LIN {X 0.035,Y -406.646,Z 971.492,A 0.000,B 0.000,C 90.000,E1 268.568} C_DIS
LIN {X -0.087,Y -402.210,Z 971.492,A 0.000,B 0.000,C 90.000,E1 268.568} C_DIS
LIN {X -0.066,Y -181.223,Z 971.492,A 0.000,B 0.000,C 90.000,E1 268.568} C_DIS
LIN {X 0.036,Y -180.887,Z 971.473,A 0.000,B 0.000,C 90.000,E1 265.122} C_DIS
LIN {X -0.082,Y -179.009,Z 971.445,A 0.000,B 0.000,C 90.000,E1 260.095} C_DIS
LIN {X 0.013,Y -178.623,Z 971.440,A 0.000,B 0.000,C 90.000,E1 259.218} C_DIS
LIN {X -0.088,Y -175.674,Z 971.412,A 0.000,B 0.000,C 90.000,E1 254.157} C_DIS
LIN {X -0.076,Y -172.391,Z 971.388,A 0.000,B 0.000,C 90.000,E1 249.880} C_DIS
LIN {X -0.060,Y -171.196,Z 971.379,A 0.000,B 0.000,C 90.000,E1 248.156} C_DIS
LIN {X -0.008,Y -167.485,Z 971.355,A 0.000,B 0.000,C 90.000,E1 243.819} C_DIS
LIN {X 0.000,Y -166.882,Z 971.350,A 0.000,B 0.000,C 90.000,E1 242.948} C_DIS
LIN {X -0.009,Y -162.187,Z 971.321,A 0.000,B 0.000,C 90.000,E1 237.709} C_DIS
LIN {X -0.042,Y -160.756,Z 971.311,A 0.000,B 0.000,C 90.000,E1 235.960} C_DIS
LIN {X 0.027,Y -157.553,Z 971.291,A 0.000,B 0.000,C 90.000,E1 232.396} C_DIS
LIN {X -0.035,Y -155.582,Z 971.276,A 0.000,B 0.000,C 90.000,E1 229.747} C_DIS
LIN {X 0.017,Y -151.866,Z 971.251,A 0.000,B 0.000,C 90.000,E1 225.243} C_DIS
LIN {X 0.030,Y -150.090,Z 971.236,A 0.000,B 0.000,C 90.000,E1 222.528} C_DIS
LIN {X -0.052,Y -146.891,Z 971.211,A 0.000,B 0.000,C 90.000,E1 218.016} C_DIS
LIN {X 0.053,Y -145.478,Z 971.196,A 0.000,B 0.000,C 90.000,E1 215.231} C_DIS
LIN {X -0.031,Y -142.888,Z 971.170,A 0.000,B 0.000,C 90.000,E1 210.669} C_DIS
LIN {X 0.026,Y -141.507,Z 971.150,A 0.000,B 0.000,C 90.000,E1 206.950} C_DIS
LIN {X -0.056,Y -139.391,Z 971.114,A 0.000,B 0.000,C 90.000,E1 200.482} C_DIS
LIN {X -0.005,Y -139.098,Z 971.103,A 0.000,B 0.000,C 90.000,E1 198.598} C_DIS
LIN {X -0.014,Y -138.353,Z 971.057,A 0.000,B 0.000,C 90.000,E1 190.197} C_DIS
LIN {X -0.020,Y -139.515,Z 971.005,A 0.000,B 0.000,C 90.000,E1 180.859} C_DIS
LIN {X 0.060,Y -141.167,Z 970.974,A 0.000,B 0.000,C 90.000,E1 175.241} C_DIS
LIN {X 0.032,Y -142.546,Z 970.958,A 0.000,B 0.000,C 90.000,E1 172.470} C_DIS
LIN {X -0.042,Y -144.821,Z 970.933,A 0.000,B 0.000,C 90.000,E1 167.881} C_DIS
LIN {X -0.056,Y -147.443,Z 970.912,A 0.000,B 0.000,C 90.000,E1 164.212} C_DIS
LIN {X -0.027,Y -150.023,Z 970.892,A 0.000,B 0.000,C 90.000,E1 160.550} C_DIS
LIN {X -0.021,Y -153.358,Z 970.872,A 0.000,B 0.000,C 90.000,E1 156.922} C_DIS
LIN {X 0.027,Y -155.892,Z 970.857,A 0.000,B 0.000,C 90.000,E1 154.204} C_DIS
LIN {X -0.075,Y -159.750,Z 970.837,A 0.000,B 0.000,C 90.000,E1 150.667} C_DIS
LIN {X -0.009,Y -161.990,Z 970.827,A 0.000,B 0.000,C 90.000,E1 148.869} C_DIS
LIN {X 0.011,Y -166.182,Z 970.807,A 0.000,B 0.000,C 90.000,E1 145.341} C_DIS
LIN {X 0.003,Y -171.197,Z 970.788,A 0.000,B 0.000,C 90.000,E1 141.859} C_DIS
LIN {X 0.033,Y -176.080,Z 970.769,A 0.000,B 0.000,C 90.000,E1 138.405} C_DIS
LIN {X -0.104,Y -180.340,Z 970.755,A 0.000,B 0.000,C 90.000,E1 135.891} C_DIS
LIN {X 0.004,Y -185.750,Z 970.736,A 0.000,B 0.000,C 90.000,E1 132.486} C_DIS
LIN {X -0.082,Y -190.362,Z 970.722,A 0.000,B 0.000,C 90.000,E1 130.011} C_DIS
LIN {X -0.069,Y -195.145,Z 970.707,A 0.000,B 0.000,C 90.000,E1 127.237} C_DIS
LIN {X -0.152,Y -298.444,Z 970.707,A 0.000,B 0.000,C 90.000,E1 127.237} C_DIS
LIN {X 0.125,Y -300.189,Z 970.707,A 0.000,B 0.000,C 90.000,E1 127.156} C_DIS
LIN {X -0.078,Y -305.216,Z 970.705,A 0.000,B 0.000,C 90.000,E1 126.950} C_DIS
LIN {X 0.147,Y -307.899,Z 970.704,A 0.000,B 0.000,C 90.000,E1 126.664} C_DIS
LIN {X -0.023,Y -311.652,Z 970.701,A 0.000,B 0.000,C 90.000,E1 126.171} C_DIS
LIN {X -0.057,Y -313.281,Z 970.699,A 0.000,B 0.000,C 90.000,E1 125.851} C_DIS
LIN {X -0.020,Y -314.559,Z 970.697,A 0.000,B 0.000,C 90.000,E1 125.518} C_DIS
LIN {X -0.088,Y -326.270,Z 970.678,A 0.000,B 0.000,C 90.000,E1 122.005} C_DIS
LIN {X 0.038,Y -337.255,Z 970.662,A 0.000,B 0.000,C 90.000,E1 119.155} C_DIS
LIN {X 0.165,Y -349.630,Z 970.647,A 0.000,B 0.000,C 90.000,E1 116.360} C_DIS
LIN {X 0.178,Y -363.508,Z 970.632,A 0.000,B 0.000,C 90.000,E1 113.643} C_DIS
LIN {X 0.187,Y -377.204,Z 970.618,A 0.000,B 0.000,C 90.000,E1 111.280} C_DIS
LIN {X -0.107,Y -392.279,Z 970.606,A 0.000,B 0.000,C 90.000,E1 109.014} C_DIS
LIN {X 0.084,Y -408.843,Z 970.593,A 0.000,B 0.000,C 90.000,E1 106.732} C_DIS
LIN {X 0.073,Y -427.015,Z 970.581,A 0.000,B 0.000,C 90.000,E1 104.537} C_DIS
LIN {X 0.151,Y -446.708,Z 970.569,A 0.000,B 0.000,C 90.000,E1 102.411} C_DIS
LIN {X -0.068,Y -467.052,Z 970.558,A 0.000,B 0.000,C 90.000,E1 100.489} C_DIS
LIN {X -0.062,Y -469.165,Z 970.557,A 0.000,B 0.000,C 90.000,E1 100.254} C_DIS
LIN {X -0.057,Y -470.766,Z 970.556,A 0.000,B 0.000,C 90.000,E1 100.018} C_DIS
LIN {X 0.261,Y -472.078,Z 970.554,A 0.000,B 0.000,C 90.000,E1 99.726} C_DIS
LIN {X 0.034,Y -473.047,Z 970.553,A 0.000,B 0.000,C 90.000,E1 99.500} C_DIS
LIN {X 0.219,Y -474.135,Z 970.550,A 0.000,B 0.000,C 90.000,E1 98.973} C_DIS
LIN {X -0.132,Y -474.233,Z 970.547,A 0.000,B 0.000,C 90.000,E1 98.511} C_DIS
LIN {X -0.007,Y -473.359,Z 970.544,A 0.000,B 0.000,C 90.000,E1 97.992} C_DIS
LIN {X 0.121,Y -471.370,Z 970.542,A 0.000,B 0.000,C 90.000,E1 97.473} C_DIS
LIN {X -0.164,Y -468.113,Z 970.539,A 0.000,B 0.000,C 90.000,E1 97.004} C_DIS
LIN {X 0.071,Y -454.642,Z 970.527,A 0.000,B 0.000,C 90.000,E1 94.935} C_DIS
LIN {X -0.006,Y -441.028,Z 970.516,A 0.000,B 0.000,C 90.000,E1 92.865} C_DIS
LIN {X 0.133,Y -426.286,Z 970.503,A 0.000,B 0.000,C 90.000,E1 90.458} C_DIS
LIN {X -0.094,Y -412.655,Z 970.489,A 0.000,B 0.000,C 90.000,E1 88.051} C_DIS
LIN {X -0.026,Y -403.632,Z 970.480,A 0.000,B 0.000,C 90.000,E1 86.388} C_DIS
LIN {X -0.040,Y -392.927,Z 970.469,A 0.000,B 0.000,C 90.000,E1 84.432} C_DIS
LIN {X 0.117,Y -383.619,Z 970.460,A 0.000,B 0.000,C 90.000,E1 82.704} C_DIS
LIN {X 0.192,Y -375.672,Z 970.452,A 0.000,B 0.000,C 90.000,E1 81.254} C_DIS
LIN {X 0.119,Y -364.228,Z 970.440,A 0.000,B 0.000,C 90.000,E1 79.218} C_DIS
LIN {X -0.119,Y -352.438,Z 970.429,A 0.000,B 0.000,C 90.000,E1 77.173} C_DIS
LIN {X 0.005,Y -334.406,Z 970.410,A 0.000,B 0.000,C 90.000,E1 73.795} C_DIS
LIN {X 0.084,Y -322.122,Z 970.396,A 0.000,B 0.000,C 90.000,E1 71.275} C_DIS
LIN {X -0.148,Y -311.513,Z 970.384,A 0.000,B 0.000,C 90.000,E1 69.082} C_DIS
LIN {X 0.077,Y -299.564,Z 970.369,A 0.000,B 0.000,C 90.000,E1 66.433} C_DIS
LIN {X 0.082,Y -287.783,Z 970.354,A 0.000,B 0.000,C 90.000,E1 63.768} C_DIS
LIN {X 0.102,Y -277.508,Z 970.341,A 0.000,B 0.000,C 90.000,E1 61.385} C_DIS
LIN {X 0.083,Y -266.012,Z 970.326,A 0.000,B 0.000,C 90.000,E1 58.614} C_DIS
LIN {X -0.021,Y -254.922,Z 970.310,A 0.000,B 0.000,C 90.000,E1 55.801} C_DIS
LIN {X -0.099,Y -243.035,Z 970.292,A 0.000,B 0.000,C 90.000,E1 52.557} C_DIS
LIN {X 0.074,Y -232.031,Z 970.273,A 0.000,B 0.000,C 90.000,E1 49.175} C_DIS
LIN {X -0.120,Y -221.821,Z 970.254,A 0.000,B 0.000,C 90.000,E1 45.810} C_DIS
LIN {X -0.005,Y -213.311,Z 970.237,A 0.000,B 0.000,C 90.000,E1 42.690} C_DIS
LIN {X -0.070,Y -205.336,Z 970.220,A 0.000,B 0.000,C 90.000,E1 39.564} C_DIS
LIN {X -0.111,Y -197.993,Z 970.202,A 0.000,B 0.000,C 90.000,E1 36.377} C_DIS
LIN {X 0.027,Y -191.300,Z 970.184,A 0.000,B 0.000,C 90.000,E1 33.086} C_DIS
LIN {X 0.004,Y -185.309,Z 970.166,A 0.000,B 0.000,C 90.000,E1 29.795} C_DIS
LIN {X 0.049,Y -180.063,Z 970.147,A 0.000,B 0.000,C 90.000,E1 26.437} C_DIS
LIN {X -0.026,Y -175.534,Z 970.128,A 0.000,B 0.000,C 90.000,E1 23.078} C_DIS
LIN {X 0.064,Y -171.707,Z 970.109,A 0.000,B 0.000,C 90.000,E1 19.631} C_DIS
LIN {X -0.096,Y -167.927,Z 970.085,A 0.000,B 0.000,C 90.000,E1 15.371} C_DIS
LIN {X -0.056,Y -165.174,Z 970.061,A 0.000,B 0.000,C 90.000,E1 11.007} C_DIS
LIN {X -0.067,Y -163.070,Z 970.027,A 0.000,B 0.000,C 90.000,E1 4.878} C_DIS
LIN {X -0.042,Y -164.371,Z 969.963,A 0.000,B 0.000,C 90.000,E1 353.394} C_DIS
LIN {X 0.037,Y -167.337,Z 969.934,A 0.000,B 0.000,C 90.000,E1 348.117} C_DIS
LIN {X 0.069,Y -170.198,Z 969.915,A 0.000,B 0.000,C 90.000,E1 344.629} C_DIS
LIN {X -0.066,Y -173.819,Z 969.896,A 0.000,B 0.000,C 90.000,E1 341.221} C_DIS
LIN {X -0.058,Y -178.179,Z 969.877,A 0.000,B 0.000,C 90.000,E1 337.794} C_DIS
LIN {X -0.067,Y -183.323,Z 969.858,A 0.000,B 0.000,C 90.000,E1 334.409} C_DIS
LIN {X -0.037,Y -189.184,Z 969.839,A 0.000,B 0.000,C 90.000,E1 331.051} C_DIS
LIN {X -0.009,Y -195.645,Z 969.821,A 0.000,B 0.000,C 90.000,E1 327.740} C_DIS
LIN {X -0.001,Y -202.711,Z 969.803,A 0.000,B 0.000,C 90.000,E1 324.482} C_DIS
LIN {X -0.010,Y -211.317,Z 969.783,A 0.000,B 0.000,C 90.000,E1 320.884} C_DIS
LIN {X -0.142,Y -220.576,Z 969.763,A 0.000,B 0.000,C 90.000,E1 317.391} C_DIS
LIN {X 0.031,Y -229.759,Z 969.746,A 0.000,B 0.000,C 90.000,E1 314.271} C_DIS
LIN {X 0.045,Y -237.519,Z 969.733,A 0.000,B 0.000,C 90.000,E1 312.000} C_DIS
LIN {X 0.047,Y -246.307,Z 969.721,A 0.000,B 0.000,C 90.000,E1 309.769} C_DIS
LIN {X 0.072,Y -254.422,Z 969.711,A 0.000,B 0.000,C 90.000,E1 307.935} C_DIS
LIN {X -0.038,Y -265.321,Z 969.699,A 0.000,B 0.000,C 90.000,E1 305.804} C_DIS
LIN {X -0.069,Y -281.207,Z 969.683,A 0.000,B 0.000,C 90.000,E1 303.007} C_DIS
LIN {X 0.092,Y -300.564,Z 969.666,A 0.000,B 0.000,C 90.000,E1 299.922} C_DIS
LIN {X -0.055,Y -314.475,Z 969.655,A 0.000,B 0.000,C 90.000,E1 297.975} C_DIS
LIN {X -0.079,Y -329.831,Z 969.645,A 0.000,B 0.000,C 90.000,E1 296.052} C_DIS
LIN {X -0.113,Y -354.177,Z 969.630,A 0.000,B 0.000,C 90.000,E1 293.387} C_DIS
LIN {X 0.029,Y -370.447,Z 969.621,A 0.000,B 0.000,C 90.000,E1 291.716} C_DIS
LIN {X 0.138,Y -389.009,Z 969.611,A 0.000,B 0.000,C 90.000,E1 289.885} C_DIS
LIN {X -0.209,Y -399.660,Z 969.605,A 0.000,B 0.000,C 90.000,E1 288.906} C_DIS
LIN {X 0.200,Y -409.889,Z 969.599,A 0.000,B 0.000,C 90.000,E1 287.819} C_DIS
LIN {X -0.155,Y -420.017,Z 969.593,A 0.000,B 0.000,C 90.000,E1 286.804} C_DIS
LIN {X -0.147,Y -429.751,Z 969.587,A 0.000,B 0.000,C 90.000,E1 285.717} C_DIS
LIN {X 0.255,Y -438.913,Z 969.581,A 0.000,B 0.000,C 90.000,E1 284.592} C_DIS
LIN {X -0.190,Y -447.466,Z 969.575,A 0.000,B 0.000,C 90.000,E1 283.592} C_DIS
LIN {X 0.160,Y -457.530,Z 969.568,A 0.000,B 0.000,C 90.000,E1 282.243} C_DIS
LIN {X -0.083,Y -465.137,Z 969.562,A 0.000,B 0.000,C 90.000,E1 281.243} C_DIS
LIN {X 0.128,Y -472.224,Z 969.557,A 0.000,B 0.000,C 90.000,E1 280.197} C_DIS
LIN {X 0.091,Y -476.879,Z 969.553,A 0.000,B 0.000,C 90.000,E1 279.443} C_DIS
LIN {X 0.100,Y -480.839,Z 969.548,A 0.000,B 0.000,C 90.000,E1 278.690} C_DIS
LIN {X 0.141,Y -484.221,Z 969.544,A 0.000,B 0.000,C 90.000,E1 277.936} C_DIS
LIN {X -0.093,Y -486.124,Z 969.541,A 0.000,B 0.000,C 90.000,E1 277.466} C_DIS
LIN {X 0.093,Y -487.737,Z 969.539,A 0.000,B 0.000,C 90.000,E1 276.947} C_DIS
LIN {X -0.193,Y -489.000,Z 969.536,A 0.000,B 0.000,C 90.000,E1 276.486} C_DIS
LIN {X 0.015,Y -489.957,Z 969.533,A 0.000,B 0.000,C 90.000,E1 275.967} C_DIS
LIN {X 0.184,Y -490.489,Z 969.530,A 0.000,B 0.000,C 90.000,E1 275.454} C_DIS
LIN {X -0.081,Y -490.737,Z 969.528,A 0.000,B 0.000,C 90.000,E1 274.992} C_DIS
LIN {X 0.144,Y -490.592,Z 969.525,A 0.000,B 0.000,C 90.000,E1 274.473} C_DIS
LIN {X -0.122,Y -489.956,Z 969.522,A 0.000,B 0.000,C 90.000,E1 274.012} C_DIS
LIN {X 0.067,Y -488.830,Z 969.519,A 0.000,B 0.000,C 90.000,E1 273.498} C_DIS
LIN {X -0.204,Y -487.113,Z 969.517,A 0.000,B 0.000,C 90.000,E1 273.037} C_DIS
LIN {X -0.022,Y -484.823,Z 969.514,A 0.000,B 0.000,C 90.000,E1 272.522} C_DIS
LIN {X 0.146,Y -481.691,Z 969.511,A 0.000,B 0.000,C 90.000,E1 272.007} C_DIS
LIN {X -0.166,Y -477.763,Z 969.508,A 0.000,B 0.000,C 90.000,E1 271.547} C_DIS
LIN {X -0.033,Y -472.805,Z 969.506,A 0.000,B 0.000,C 90.000,E1 271.031} C_DIS
LIN {X -0.206,Y -466.997,Z 969.503,A 0.000,B 0.000,C 90.000,E1 270.573} C_DIS
LIN {X 0.051,Y -460.783,Z 969.501,A 0.000,B 0.000,C 90.000,E1 270.115} C_DIS
LIN {X -0.192,Y -454.151,Z 969.499,A 0.000,B 0.000,C 90.000,E1 269.771} C_DIS
LIN {X 0.015,Y -447.184,Z 969.497,A 0.000,B 0.000,C 90.000,E1 269.427} C_DIS
LIN {X 0.193,Y -440.049,Z 969.495,A 0.000,B 0.000,C 90.000,E1 269.141} C_DIS
LIN {X -0.170,Y -432.430,Z 969.494,A 0.000,B 0.000,C 90.000,E1 268.969} C_DIS
LIN {X -0.149,Y -424.534,Z 969.493,A 0.000,B 0.000,C 90.000,E1 268.797} C_DIS
LIN {X 0.166,Y -416.590,Z 969.492,A 0.000,B 0.000,C 90.000,E1 268.625} C_DIS
LIN {X 0.033,Y -409.424,Z 969.492,A 0.000,B 0.000,C 90.000,E1 268.568} C_DIS
LIN {X -0.198,Y -403.286,Z 969.492,A 0.000,B 0.000,C 90.000,E1 268.568} C_DIS
LIN {X 0.068,Y -181.220,Z 969.492,A 0.000,B 0.000,C 90.000,E1 268.511} C_DIS
LIN {X -0.021,Y -180.884,Z 969.473,A 0.000,B 0.000,C 90.000,E1 265.122} C_DIS
LIN {X 0.039,Y -179.005,Z 969.445,A 0.000,B 0.000,C 90.000,E1 260.038} C_DIS
LIN {X -0.043,Y -178.610,Z 969.440,A 0.000,B 0.000,C 90.000,E1 259.218} C_DIS
LIN {X 0.026,Y -175.662,Z 969.412,A 0.000,B 0.000,C 90.000,E1 254.102} C_DIS
LIN {X 0.030,Y -172.379,Z 969.388,A 0.000,B 0.000,C 90.000,E1 249.826} C_DIS
LIN {X 0.044,Y -171.177,Z 969.378,A 0.000,B 0.000,C 90.000,E1 248.103} C_DIS
LIN {X 0.088,Y -167.472,Z 969.354,A 0.000,B 0.000,C 90.000,E1 243.768} C_DIS
LIN {X 0.021,Y -166.868,Z 969.350,A 0.000,B 0.000,C 90.000,E1 242.922} C_DIS
LIN {X 0.075,Y -162.173,Z 969.320,A 0.000,B 0.000,C 90.000,E1 237.661} C_DIS
LIN {X -0.005,Y -160.736,Z 969.311,A 0.000,B 0.000,C 90.000,E1 235.928} C_DIS
LIN {X -0.026,Y -157.538,Z 969.291,A 0.000,B 0.000,C 90.000,E1 232.396} C_DIS
LIN {X 0.032,Y -155.564,Z 969.276,A 0.000,B 0.000,C 90.000,E1 229.703} C_DIS
LIN {X -0.034,Y -151.853,Z 969.251,A 0.000,B 0.000,C 90.000,E1 225.243} C_DIS
LIN {X -0.020,Y -150.074,Z 969.236,A 0.000,B 0.000,C 90.000,E1 222.528} C_DIS
LIN {X 0.014,Y -146.880,Z 969.211,A 0.000,B 0.000,C 90.000,E1 217.971} C_DIS
LIN {X 0.003,Y -145.466,Z 969.196,A 0.000,B 0.000,C 90.000,E1 215.231} C_DIS
LIN {X -0.079,Y -142.879,Z 969.170,A 0.000,B 0.000,C 90.000,E1 210.669} C_DIS
LIN {X -0.023,Y -141.497,Z 969.150,A 0.000,B 0.000,C 90.000,E1 206.950} C_DIS
LIN {X 0.026,Y -139.387,Z 969.114,A 0.000,B 0.000,C 90.000,E1 200.429} C_DIS
LIN {X 0.014,Y -138.844,Z 969.098,A 0.000,B 0.000,C 90.000,E1 197.638} C_DIS
LIN {X -0.062,Y -138.353,Z 969.057,A 0.000,B 0.000,C 90.000,E1 190.197} C_DIS
LIN {X -0.070,Y -139.518,Z 969.005,A 0.000,B 0.000,C 90.000,E1 180.859} C_DIS
LIN {X 0.011,Y -141.176,Z 968.974,A 0.000,B 0.000,C 90.000,E1 175.241} C_DIS
LIN {X -0.017,Y -142.555,Z 968.958,A 0.000,B 0.000,C 90.000,E1 172.470} C_DIS
LIN {X 0.050,Y -144.833,Z 968.932,A 0.000,B 0.000,C 90.000,E1 167.825} C_DIS
LIN {X 0.036,Y -147.455,Z 968.912,A 0.000,B 0.000,C 90.000,E1 164.157} C_DIS
LIN {X -0.078,Y -150.039,Z 968.892,A 0.000,B 0.000,C 90.000,E1 160.550} C_DIS
LIN {X -0.072,Y -153.378,Z 968.872,A 0.000,B 0.000,C 90.000,E1 156.922} C_DIS
LIN {X -0.024,Y -155.910,Z 968.857,A 0.000,B 0.000,C 90.000,E1 154.204} C_DIS
LIN {X 0.090,Y -159.773,Z 968.837,A 0.000,B 0.000,C 90.000,E1 150.589} C_DIS
LIN {X -0.062,Y -162.014,Z 968.827,A 0.000,B 0.000,C 90.000,E1 148.869} C_DIS
LIN {X 0.052,Y -166.208,Z 968.807,A 0.000,B 0.000,C 90.000,E1 145.308} C_DIS
LIN {X 0.054,Y -171.223,Z 968.788,A 0.000,B 0.000,C 90.000,E1 141.823} C_DIS
LIN {X -0.022,Y -176.108,Z 968.769,A 0.000,B 0.000,C 90.000,E1 138.405} C_DIS
LIN {X 0.094,Y -180.372,Z 968.755,A 0.000,B 0.000,C 90.000,E1 135.810} C_DIS
LIN {X 0.072,Y -185.780,Z 968.736,A 0.000,B 0.000,C 90.000,E1 132.447} C_DIS
LIN {X 0.005,Y -190.396,Z 968.722,A 0.000,B 0.000,C 90.000,E1 129.967} C_DIS
LIN {X 0.030,Y -195.092,Z 968.707,A 0.000,B 0.000,C 90.000,E1 127.237} C_DIS
LIN {X -0.004,Y -298.842,Z 968.707,A 0.000,B 0.000,C 90.000,E1 127.237} C_DIS
LIN {X 0.000,Y -305.337,Z 968.705,A 0.000,B 0.000,C 90.000,E1 126.950} C_DIS
LIN {X 0.053,Y -308.226,Z 968.704,A 0.000,B 0.000,C 90.000,E1 126.664} C_DIS
LIN {X -0.047,Y -311.919,Z 968.701,A 0.000,B 0.000,C 90.000,E1 126.137} C_DIS
LIN {X -0.010,Y -313.464,Z 968.699,A 0.000,B 0.000,C 90.000,E1 125.804} C_DIS
LIN {X 0.028,Y -314.678,Z 968.697,A 0.000,B 0.000,C 90.000,E1 125.471} C_DIS
LIN {X 0.048,Y -325.248,Z 968.679,A 0.000,B 0.000,C 90.000,E1 122.260} C_DIS
LIN {X 0.145,Y -336.099,Z 968.664,A 0.000,B 0.000,C 90.000,E1 119.411} C_DIS
LIN {X -0.075,Y -348.336,Z 968.648,A 0.000,B 0.000,C 90.000,E1 116.668} C_DIS
LIN {X -0.110,Y -362.059,Z 968.633,A 0.000,B 0.000,C 90.000,E1 113.951} C_DIS
LIN {X -0.150,Y -375.608,Z 968.620,A 0.000,B 0.000,C 90.000,E1 111.589} C_DIS
LIN {X -0.124,Y -390.526,Z 968.607,A 0.000,B 0.000,C 90.000,E1 109.268} C_DIS
LIN {X 0.030,Y -406.921,Z 968.594,A 0.000,B 0.000,C 90.000,E1 106.985} C_DIS
LIN {X 0.091,Y -424.908,Z 968.582,A 0.000,B 0.000,C 90.000,E1 104.773} C_DIS
LIN {X 0.067,Y -444.470,Z 968.570,A 0.000,B 0.000,C 90.000,E1 102.647} C_DIS
LIN {X 0.155,Y -467.321,Z 968.558,A 0.000,B 0.000,C 90.000,E1 100.433} C_DIS
LIN {X 0.154,Y -469.373,Z 968.557,A 0.000,B 0.000,C 90.000,E1 100.197} C_DIS
LIN {X 0.152,Y -470.931,Z 968.555,A 0.000,B 0.000,C 90.000,E1 99.962} C_DIS
LIN {X 0.005,Y -472.201,Z 968.554,A 0.000,B 0.000,C 90.000,E1 99.726} C_DIS
LIN {X -0.221,Y -473.134,Z 968.553,A 0.000,B 0.000,C 90.000,E1 99.500} C_DIS
LIN {X -0.034,Y -474.164,Z 968.550,A 0.000,B 0.000,C 90.000,E1 98.973} C_DIS
LIN {X 0.083,Y -474.208,Z 968.547,A 0.000,B 0.000,C 90.000,E1 98.454} C_DIS
LIN {X 0.209,Y -473.277,Z 968.544,A 0.000,B 0.000,C 90.000,E1 97.936} C_DIS
LIN {X -0.070,Y -471.217,Z 968.541,A 0.000,B 0.000,C 90.000,E1 97.466} C_DIS
LIN {X -0.070,Y -462.876,Z 968.534,A 0.000,B 0.000,C 90.000,E1 96.201} C_DIS
LIN {X -0.157,Y -451.081,Z 968.524,A 0.000,B 0.000,C 90.000,E1 94.416} C_DIS
LIN {X 0.104,Y -437.534,Z 968.513,A 0.000,B 0.000,C 90.000,E1 92.293} C_DIS
LIN {X -0.143,Y -421.551,Z 968.498,A 0.000,B 0.000,C 90.000,E1 89.656} C_DIS
LIN {X -0.155,Y -409.533,Z 968.486,A 0.000,B 0.000,C 90.000,E1 87.478} C_DIS
LIN {X -0.076,Y -398.906,Z 968.475,A 0.000,B 0.000,C 90.000,E1 85.527} C_DIS
LIN {X -0.185,Y -388.138,Z 968.464,A 0.000,B 0.000,C 90.000,E1 83.571} C_DIS
LIN {X -0.069,Y -378.742,Z 968.455,A 0.000,B 0.000,C 90.000,E1 81.837} C_DIS
LIN {X -0.067,Y -368.980,Z 968.445,A 0.000,B 0.000,C 90.000,E1 80.095} C_DIS
LIN {X -0.145,Y -360.706,Z 968.437,A 0.000,B 0.000,C 90.000,E1 78.634} C_DIS
LIN {X -0.028,Y -348.897,Z 968.425,A 0.000,B 0.000,C 90.000,E1 76.520} C_DIS
LIN {X 0.005,Y -332.693,Z 968.408,A 0.000,B 0.000,C 90.000,E1 73.449} C_DIS
LIN {X 0.136,Y -320.467,Z 968.394,A 0.000,B 0.000,C 90.000,E1 70.913} C_DIS
LIN {X -0.139,Y -309.852,Z 968.382,A 0.000,B 0.000,C 90.000,E1 68.720} C_DIS
LIN {X -0.001,Y -299.423,Z 968.369,A 0.000,B 0.000,C 90.000,E1 66.410} C_DIS
LIN {X 0.028,Y -289.087,Z 968.356,A 0.000,B 0.000,C 90.000,E1 64.076} C_DIS
LIN {X -0.043,Y -278.808,Z 968.343,A 0.000,B 0.000,C 90.000,E1 61.719} C_DIS
LIN {X -0.026,Y -267.251,Z 968.327,A 0.000,B 0.000,C 90.000,E1 58.948} C_DIS
LIN {X 0.118,Y -256.104,Z 968.312,A 0.000,B 0.000,C 90.000,E1 56.087} C_DIS
LIN {X 0.060,Y -244.147,Z 968.294,A 0.000,B 0.000,C 90.000,E1 52.844} C_DIS
LIN {X -0.066,Y -233.081,Z 968.275,A 0.000,B 0.000,C 90.000,E1 49.542} C_DIS
LIN {X 0.002,Y -223.919,Z 968.258,A 0.000,B 0.000,C 90.000,E1 46.500} C_DIS
LIN {X 0.016,Y -215.320,Z 968.241,A 0.000,B 0.000,C 90.000,E1 43.419} C_DIS
LIN {X -0.018,Y -207.225,Z 968.224,A 0.000,B 0.000,C 90.000,E1 40.297} C_DIS
LIN {X 0.104,Y -199.753,Z 968.206,A 0.000,B 0.000,C 90.000,E1 37.076} C_DIS
LIN {X 0.011,Y -192.913,Z 968.188,A 0.000,B 0.000,C 90.000,E1 33.865} C_DIS
LIN {X -0.031,Y -186.759,Z 968.170,A 0.000,B 0.000,C 90.000,E1 30.590} C_DIS
LIN {X -0.026,Y -181.363,Z 968.151,A 0.000,B 0.000,C 90.000,E1 27.257} C_DIS
LIN {X -0.070,Y -176.653,Z 968.133,A 0.000,B 0.000,C 90.000,E1 23.898} C_DIS
LIN {X -0.047,Y -172.680,Z 968.114,A 0.000,B 0.000,C 90.000,E1 20.482} C_DIS
LIN {X 0.036,Y -168.694,Z 968.090,A 0.000,B 0.000,C 90.000,E1 16.150} C_DIS
LIN {X -0.022,Y -165.740,Z 968.066,A 0.000,B 0.000,C 90.000,E1 11.827} C_DIS
LIN {X 0.032,Y -163.352,Z 968.032,A 0.000,B 0.000,C 90.000,E1 5.682} C_DIS
LIN {X -0.036,Y -164.525,Z 967.963,A 0.000,B 0.000,C 90.000,E1 353.394} C_DIS
LIN {X 0.050,Y -167.494,Z 967.934,A 0.000,B 0.000,C 90.000,E1 348.117} C_DIS
LIN {X 0.085,Y -170.394,Z 967.915,A 0.000,B 0.000,C 90.000,E1 344.629} C_DIS
LIN {X -0.045,Y -174.011,Z 967.896,A 0.000,B 0.000,C 90.000,E1 341.221} C_DIS
LIN {X -0.031,Y -178.375,Z 967.877,A 0.000,B 0.000,C 90.000,E1 337.794} C_DIS
LIN {X -0.035,Y -183.524,Z 967.858,A 0.000,B 0.000,C 90.000,E1 334.409} C_DIS
LIN {X 0.001,Y -189.365,Z 967.839,A 0.000,B 0.000,C 90.000,E1 331.051} C_DIS
LIN {X 0.035,Y -195.821,Z 967.821,A 0.000,B 0.000,C 90.000,E1 327.740} C_DIS
LIN {X 0.049,Y -202.881,Z 967.803,A 0.000,B 0.000,C 90.000,E1 324.482} C_DIS
LIN {X 0.048,Y -211.490,Z 967.783,A 0.000,B 0.000,C 90.000,E1 320.884} C_DIS
LIN {X -0.078,Y -220.774,Z 967.763,A 0.000,B 0.000,C 90.000,E1 317.391} C_DIS
LIN {X 0.104,Y -229.962,Z 967.746,A 0.000,B 0.000,C 90.000,E1 314.271} C_DIS
LIN {X -0.052,Y -237.716,Z 967.734,A 0.000,B 0.000,C 90.000,E1 312.043} C_DIS
LIN {X -0.026,Y -248.010,Z 967.719,A 0.000,B 0.000,C 90.000,E1 309.439} C_DIS
LIN {X 0.026,Y -256.288,Z 967.709,A 0.000,B 0.000,C 90.000,E1 307.604} C_DIS
LIN {X 0.018,Y -269.252,Z 967.695,A 0.000,B 0.000,C 90.000,E1 305.105} C_DIS
LIN {X -0.103,Y -287.543,Z 967.678,A 0.000,B 0.000,C 90.000,E1 302.005} C_DIS
LIN {X 0.107,Y -307.324,Z 967.661,A 0.000,B 0.000,C 90.000,E1 298.949} C_DIS
LIN {X 0.096,Y -321.891,Z 967.650,A 0.000,B 0.000,C 90.000,E1 297.001} C_DIS
LIN {X -0.070,Y -337.700,Z 967.640,A 0.000,B 0.000,C 90.000,E1 295.155} C_DIS
LIN {X -0.068,Y -362.118,Z 967.625,A 0.000,B 0.000,C 90.000,E1 292.567} C_DIS
LIN {X 0.120,Y -380.925,Z 967.615,A 0.000,B 0.000,C 90.000,E1 290.663} C_DIS
LIN {X -0.112,Y -396.946,Z 967.606,A 0.000,B 0.000,C 90.000,E1 289.141} C_DIS
LIN {X -0.058,Y -404.749,Z 967.602,A 0.000,B 0.000,C 90.000,E1 288.362} C_DIS
LIN {X 0.172,Y -414.993,Z 967.596,A 0.000,B 0.000,C 90.000,E1 287.275} C_DIS
LIN {X -0.024,Y -422.506,Z 967.592,A 0.000,B 0.000,C 90.000,E1 286.496} C_DIS
LIN {X -0.111,Y -432.077,Z 967.586,A 0.000,B 0.000,C 90.000,E1 285.426} C_DIS
LIN {X 0.122,Y -438.893,Z 967.581,A 0.000,B 0.000,C 90.000,E1 284.592} C_DIS
LIN {X -0.094,Y -449.460,Z 967.574,A 0.000,B 0.000,C 90.000,E1 283.300} C_DIS
LIN {X -0.165,Y -459.422,Z 967.567,A 0.000,B 0.000,C 90.000,E1 282.007} C_DIS
LIN {X 0.065,Y -466.926,Z 967.561,A 0.000,B 0.000,C 90.000,E1 280.950} C_DIS
LIN {X -0.018,Y -472.208,Z 967.557,A 0.000,B 0.000,C 90.000,E1 280.197} C_DIS
LIN {X -0.057,Y -476.903,Z 967.552,A 0.000,B 0.000,C 90.000,E1 279.443} C_DIS
LIN {X 0.023,Y -480.876,Z 967.548,A 0.000,B 0.000,C 90.000,E1 278.681} C_DIS
LIN {X -0.009,Y -484.299,Z 967.544,A 0.000,B 0.000,C 90.000,E1 277.936} C_DIS
LIN {X 0.238,Y -486.207,Z 967.541,A 0.000,B 0.000,C 90.000,E1 277.409} C_DIS
LIN {X -0.057,Y -487.811,Z 967.539,A 0.000,B 0.000,C 90.000,E1 276.947} C_DIS
LIN {X 0.143,Y -489.062,Z 967.536,A 0.000,B 0.000,C 90.000,E1 276.429} C_DIS
LIN {X -0.136,Y -490.002,Z 967.533,A 0.000,B 0.000,C 90.000,E1 275.967} C_DIS
LIN {X 0.034,Y -490.584,Z 967.530,A 0.000,B 0.000,C 90.000,E1 275.454} C_DIS
LIN {X -0.231,Y -490.821,Z 967.528,A 0.000,B 0.000,C 90.000,E1 274.992} C_DIS
LIN {X -0.005,Y -490.647,Z 967.525,A 0.000,B 0.000,C 90.000,E1 274.473} C_DIS
LIN {X 0.219,Y -489.998,Z 967.522,A 0.000,B 0.000,C 90.000,E1 273.955} C_DIS
LIN {X -0.080,Y -488.863,Z 967.519,A 0.000,B 0.000,C 90.000,E1 273.498} C_DIS
LIN {X 0.135,Y -487.149,Z 967.517,A 0.000,B 0.000,C 90.000,E1 272.980} C_DIS
LIN {X -0.167,Y -484.810,Z 967.514,A 0.000,B 0.000,C 90.000,E1 272.522} C_DIS
LIN {X 0.002,Y -481.707,Z 967.511,A 0.000,B 0.000,C 90.000,E1 272.007} C_DIS
LIN {X 0.168,Y -477.738,Z 967.508,A 0.000,B 0.000,C 90.000,E1 271.489} C_DIS
LIN {X -0.005,Y -475.385,Z 967.507,A 0.000,B 0.000,C 90.000,E1 271.260} C_DIS
LIN {X 0.231,Y -469.969,Z 967.504,A 0.000,B 0.000,C 90.000,E1 270.745} C_DIS
LIN {X 0.164,Y -466.996,Z 967.503,A 0.000,B 0.000,C 90.000,E1 270.516} C_DIS
LIN {X -0.049,Y -460.751,Z 967.501,A 0.000,B 0.000,C 90.000,E1 270.115} C_DIS
LIN {X 0.135,Y -454.096,Z 967.498,A 0.000,B 0.000,C 90.000,E1 269.714} C_DIS
LIN {X -0.087,Y -447.192,Z 967.497,A 0.000,B 0.000,C 90.000,E1 269.427} C_DIS
LIN {X 0.109,Y -440.205,Z 967.495,A 0.000,B 0.000,C 90.000,E1 269.141} C_DIS
LIN {X 0.186,Y -432.679,Z 967.494,A 0.000,B 0.000,C 90.000,E1 268.912} C_DIS
LIN {X 0.187,Y -424.857,Z 967.493,A 0.000,B 0.000,C 90.000,E1 268.740} C_DIS
LIN {X 0.053,Y -416.867,Z 967.492,A 0.000,B 0.000,C 90.000,E1 268.625} C_DIS
LIN {X -0.085,Y -409.839,Z 967.492,A 0.000,B 0.000,C 90.000,E1 268.568} C_DIS
LIN {X 0.085,Y -404.035,Z 967.492,A 0.000,B 0.000,C 90.000,E1 268.511} C_DIS
LIN {X 0.031,Y -397.395,Z 967.492,A 0.000,B 0.000,C 90.000,E1 268.511} C_DIS
LIN {X -0.010,Y -181.215,Z 967.492,A 0.000,B 0.000,C 90.000,E1 268.511} C_DIS
LIN {X -0.074,Y -180.881,Z 967.473,A 0.000,B 0.000,C 90.000,E1 265.122} C_DIS
LIN {X -0.013,Y -179.001,Z 967.445,A 0.000,B 0.000,C 90.000,E1 260.038} C_DIS
LIN {X 0.080,Y -178.598,Z 967.440,A 0.000,B 0.000,C 90.000,E1 259.162} C_DIS
LIN {X -0.026,Y -175.650,Z 967.412,A 0.000,B 0.000,C 90.000,E1 254.102} C_DIS
LIN {X -0.020,Y -172.369,Z 967.388,A 0.000,B 0.000,C 90.000,E1 249.826} C_DIS
LIN {X -0.007,Y -171.160,Z 967.378,A 0.000,B 0.000,C 90.000,E1 248.103} C_DIS
LIN {X 0.038,Y -167.459,Z 967.354,A 0.000,B 0.000,C 90.000,E1 243.768} C_DIS
LIN {X -0.029,Y -166.855,Z 967.349,A 0.000,B 0.000,C 90.000,E1 242.922} C_DIS
LIN {X 0.036,Y -162.841,Z 967.325,A 0.000,B 0.000,C 90.000,E1 238.535} C_DIS
LIN {X 0.011,Y -161.525,Z 967.315,A 0.000,B 0.000,C 90.000,E1 236.786} C_DIS
LIN {X 0.051,Y -157.524,Z 967.291,A 0.000,B 0.000,C 90.000,E1 232.351} C_DIS
LIN {X -0.016,Y -155.549,Z 967.276,A 0.000,B 0.000,C 90.000,E1 229.703} C_DIS
LIN {X -0.081,Y -151.841,Z 967.251,A 0.000,B 0.000,C 90.000,E1 225.243} C_DIS
LIN {X -0.067,Y -150.059,Z 967.236,A 0.000,B 0.000,C 90.000,E1 222.528} C_DIS
LIN {X -0.032,Y -146.869,Z 967.211,A 0.000,B 0.000,C 90.000,E1 217.971} C_DIS
LIN {X -0.043,Y -145.455,Z 967.196,A 0.000,B 0.000,C 90.000,E1 215.231} C_DIS
LIN {X 0.070,Y -142.871,Z 967.170,A 0.000,B 0.000,C 90.000,E1 210.590} C_DIS
LIN {X -0.004,Y -141.488,Z 967.150,A 0.000,B 0.000,C 90.000,E1 206.924} C_DIS
LIN {X -0.019,Y -139.385,Z 967.113,A 0.000,B 0.000,C 90.000,E1 200.429} C_DIS
LIN {X -0.030,Y -138.839,Z 967.098,A 0.000,B 0.000,C 90.000,E1 197.638} C_DIS
LIN {X 0.030,Y -138.354,Z 967.056,A 0.000,B 0.000,C 90.000,E1 190.141} C_DIS
LIN {X 0.025,Y -139.521,Z 967.005,A 0.000,B 0.000,C 90.000,E1 180.802} C_DIS
LIN {X -0.034,Y -141.184,Z 966.974,A 0.000,B 0.000,C 90.000,E1 175.241} C_DIS
LIN {X -0.063,Y -142.562,Z 966.958,A 0.000,B 0.000,C 90.000,E1 172.470} C_DIS
LIN {X 0.003,Y -144.844,Z 966.932,A 0.000,B 0.000,C 90.000,E1 167.825} C_DIS
LIN {X -0.011,Y -147.469,Z 966.912,A 0.000,B 0.000,C 90.000,E1 164.157} C_DIS
LIN {X 0.016,Y -150.054,Z 966.892,A 0.000,B 0.000,C 90.000,E1 160.496} C_DIS
LIN {X 0.021,Y -153.397,Z 966.872,A 0.000,B 0.000,C 90.000,E1 156.869} C_DIS
LIN {X 0.068,Y -155.928,Z 966.857,A 0.000,B 0.000,C 90.000,E1 154.152} C_DIS
LIN {X 0.042,Y -159.795,Z 966.837,A 0.000,B 0.000,C 90.000,E1 150.589} C_DIS
LIN {X 0.028,Y -162.035,Z 966.827,A 0.000,B 0.000,C 90.000,E1 148.820} C_DIS
LIN {X 0.002,Y -166.230,Z 966.807,A 0.000,B 0.000,C 90.000,E1 145.308} C_DIS
LIN {X 0.003,Y -171.246,Z 966.788,A 0.000,B 0.000,C 90.000,E1 141.823} C_DIS
LIN {X -0.075,Y -176.135,Z 966.769,A 0.000,B 0.000,C 90.000,E1 138.405} C_DIS
LIN {X 0.042,Y -180.402,Z 966.755,A 0.000,B 0.000,C 90.000,E1 135.810} C_DIS
LIN {X 0.018,Y -185.810,Z 966.736,A 0.000,B 0.000,C 90.000,E1 132.447} C_DIS
LIN {X 0.073,Y -190.428,Z 966.722,A 0.000,B 0.000,C 90.000,E1 129.930} C_DIS
LIN {X 0.009,Y -195.020,Z 966.707,A 0.000,B 0.000,C 90.000,E1 127.282} C_DIS
LIN {X -0.036,Y -297.685,Z 966.707,A 0.000,B 0.000,C 90.000,E1 127.282} C_DIS
LIN {X 0.054,Y -303.133,Z 966.706,A 0.000,B 0.000,C 90.000,E1 127.111} C_DIS
LIN {X 0.086,Y -305.426,Z 966.705,A 0.000,B 0.000,C 90.000,E1 126.950} C_DIS
LIN {X -0.035,Y -308.523,Z 966.704,A 0.000,B 0.000,C 90.000,E1 126.664} C_DIS
LIN {X 0.019,Y -312.150,Z 966.701,A 0.000,B 0.000,C 90.000,E1 126.091} C_DIS
LIN {X -0.196,Y -313.617,Z 966.699,A 0.000,B 0.000,C 90.000,E1 125.804} C_DIS
LIN {X -0.121,Y -316.765,Z 966.693,A 0.000,B 0.000,C 90.000,E1 124.818} C_DIS
LIN {X 0.052,Y -327.646,Z 966.676,A 0.000,B 0.000,C 90.000,E1 121.592} C_DIS
LIN {X 0.058,Y -338.812,Z 966.660,A 0.000,B 0.000,C 90.000,E1 118.771} C_DIS
LIN {X -0.087,Y -351.386,Z 966.645,A 0.000,B 0.000,C 90.000,E1 116.027} C_DIS
LIN {X -0.183,Y -365.474,Z 966.629,A 0.000,B 0.000,C 90.000,E1 113.334} C_DIS
LIN {X -0.137,Y -379.374,Z 966.616,A 0.000,B 0.000,C 90.000,E1 110.972} C_DIS
LIN {X -0.146,Y -394.670,Z 966.604,A 0.000,B 0.000,C 90.000,E1 108.671} C_DIS
LIN {X 0.120,Y -411.471,Z 966.591,A 0.000,B 0.000,C 90.000,E1 106.386} C_DIS
LIN {X -0.229,Y -429.900,Z 966.579,A 0.000,B 0.000,C 90.000,E1 104.245} C_DIS
LIN {X 0.016,Y -449.732,Z 966.567,A 0.000,B 0.000,C 90.000,E1 102.119} C_DIS
LIN {X -0.048,Y -467.541,Z 966.558,A 0.000,B 0.000,C 90.000,E1 100.433} C_DIS
LIN {X -0.060,Y -469.547,Z 966.557,A 0.000,B 0.000,C 90.000,E1 100.197} C_DIS
LIN {X -0.074,Y -471.071,Z 966.555,A 0.000,B 0.000,C 90.000,E1 99.962} C_DIS
LIN {X 0.245,Y -472.304,Z 966.554,A 0.000,B 0.000,C 90.000,E1 99.670} C_DIS
LIN {X 0.020,Y -473.208,Z 966.552,A 0.000,B 0.000,C 90.000,E1 99.443} C_DIS
LIN {X 0.208,Y -474.187,Z 966.550,A 0.000,B 0.000,C 90.000,E1 98.916} C_DIS
LIN {X -0.143,Y -474.184,Z 966.547,A 0.000,B 0.000,C 90.000,E1 98.454} C_DIS
LIN {X -0.016,Y -473.203,Z 966.544,A 0.000,B 0.000,C 90.000,E1 97.936} C_DIS
LIN {X 0.173,Y -471.080,Z 966.541,A 0.000,B 0.000,C 90.000,E1 97.409} C_DIS
LIN {X -0.222,Y -459.382,Z 966.531,A 0.000,B 0.000,C 90.000,E1 95.682} C_DIS
LIN {X 0.070,Y -447.577,Z 966.521,A 0.000,B 0.000,C 90.000,E1 93.841} C_DIS
LIN {X -0.043,Y -432.474,Z 966.508,A 0.000,B 0.000,C 90.000,E1 91.489} C_DIS
LIN {X 0.183,Y -413.922,Z 966.490,A 0.000,B 0.000,C 90.000,E1 88.224} C_DIS
LIN {X -0.123,Y -404.884,Z 966.481,A 0.000,B 0.000,C 90.000,E1 86.617} C_DIS
LIN {X -0.138,Y -394.175,Z 966.470,A 0.000,B 0.000,C 90.000,E1 84.666} C_DIS
LIN {X 0.073,Y -383.338,Z 966.459,A 0.000,B 0.000,C 90.000,E1 82.648} C_DIS
LIN {X 0.143,Y -375.384,Z 966.451,A 0.000,B 0.000,C 90.000,E1 81.197} C_DIS
LIN {X 0.062,Y -363.914,Z 966.440,A 0.000,B 0.000,C 90.000,E1 79.162} C_DIS
LIN {X -0.134,Y -353.830,Z 966.430,A 0.000,B 0.000,C 90.000,E1 77.409} C_DIS
LIN {X 0.050,Y -337.252,Z 966.413,A 0.000,B 0.000,C 90.000,E1 74.338} C_DIS
LIN {X 0.052,Y -323.373,Z 966.397,A 0.000,B 0.000,C 90.000,E1 71.529} C_DIS
LIN {X -0.055,Y -312.762,Z 966.385,A 0.000,B 0.000,C 90.000,E1 69.316} C_DIS
LIN {X -0.070,Y -300.780,Z 966.371,A 0.000,B 0.000,C 90.000,E1 66.719} C_DIS
LIN {X 0.118,Y -288.951,Z 966.356,A 0.000,B 0.000,C 90.000,E1 64.024} C_DIS
LIN {X -0.043,Y -280.120,Z 966.345,A 0.000,B 0.000,C 90.000,E1 62.025} C_DIS
LIN {X 0.016,Y -268.509,Z 966.329,A 0.000,B 0.000,C 90.000,E1 59.253} C_DIS
LIN {X 0.020,Y -258.695,Z 966.315,A 0.000,B 0.000,C 90.000,E1 56.786} C_DIS
LIN {X 0.035,Y -246.591,Z 966.297,A 0.000,B 0.000,C 90.000,E1 53.543} C_DIS
LIN {X 0.015,Y -235.333,Z 966.279,A 0.000,B 0.000,C 90.000,E1 50.231} C_DIS
LIN {X 0.073,Y -224.940,Z 966.260,A 0.000,B 0.000,C 90.000,E1 46.824} C_DIS
LIN {X 0.010,Y -215.270,Z 966.241,A 0.000,B 0.000,C 90.000,E1 43.380} C_DIS
LIN {X -0.010,Y -207.190,Z 966.224,A 0.000,B 0.000,C 90.000,E1 40.253} C_DIS
LIN {X -0.041,Y -199.744,Z 966.206,A 0.000,B 0.000,C 90.000,E1 37.076} C_DIS
LIN {X -0.022,Y -192.946,Z 966.188,A 0.000,B 0.000,C 90.000,E1 33.833} C_DIS
LIN {X -0.005,Y -186.798,Z 966.170,A 0.000,B 0.000,C 90.000,E1 30.541} C_DIS
LIN {X 0.005,Y -181.420,Z 966.151,A 0.000,B 0.000,C 90.000,E1 27.206} C_DIS
LIN {X 0.038,Y -176.727,Z 966.132,A 0.000,B 0.000,C 90.000,E1 23.823} C_DIS
LIN {X -0.006,Y -172.758,Z 966.113,A 0.000,B 0.000,C 90.000,E1 20.429} C_DIS
LIN {X -0.033,Y -168.788,Z 966.090,A 0.000,B 0.000,C 90.000,E1 16.134} C_DIS
LIN {X 0.030,Y -165.841,Z 966.065,A 0.000,B 0.000,C 90.000,E1 11.771} C_DIS
LIN {X -0.073,Y -163.465,Z 966.031,A 0.000,B 0.000,C 90.000,E1 5.682} C_DIS
LIN {X -0.030,Y -164.683,Z 965.963,A 0.000,B 0.000,C 90.000,E1 353.394} C_DIS
LIN {X 0.062,Y -167.672,Z 965.934,A 0.000,B 0.000,C 90.000,E1 348.117} C_DIS
LIN {X -0.063,Y -170.591,Z 965.915,A 0.000,B 0.000,C 90.000,E1 344.685} C_DIS
LIN {X -0.022,Y -174.211,Z 965.896,A 0.000,B 0.000,C 90.000,E1 341.221} C_DIS
LIN {X -0.004,Y -178.578,Z 965.877,A 0.000,B 0.000,C 90.000,E1 337.794} C_DIS
LIN {X -0.001,Y -183.723,Z 965.858,A 0.000,B 0.000,C 90.000,E1 334.409} C_DIS
LIN {X 0.041,Y -189.554,Z 965.839,A 0.000,B 0.000,C 90.000,E1 331.051} C_DIS
LIN {X -0.085,Y -196.001,Z 965.821,A 0.000,B 0.000,C 90.000,E1 327.788} C_DIS
LIN {X 0.101,Y -203.063,Z 965.803,A 0.000,B 0.000,C 90.000,E1 324.482} C_DIS
LIN {X 0.107,Y -211.666,Z 965.783,A 0.000,B 0.000,C 90.000,E1 320.884} C_DIS
LIN {X -0.011,Y -220.978,Z 965.763,A 0.000,B 0.000,C 90.000,E1 317.391} C_DIS
LIN {X 0.015,Y -230.161,Z 965.746,A 0.000,B 0.000,C 90.000,E1 314.312} C_DIS
LIN {X 0.030,Y -237.915,Z 965.734,A 0.000,B 0.000,C 90.000,E1 312.043} C_DIS
LIN {X 0.063,Y -248.172,Z 965.719,A 0.000,B 0.000,C 90.000,E1 309.439} C_DIS
LIN {X -0.082,Y -256.409,Z 965.709,A 0.000,B 0.000,C 90.000,E1 307.649} C_DIS
LIN {X 0.121,Y -269.350,Z 965.695,A 0.000,B 0.000,C 90.000,E1 305.105} C_DIS
LIN {X 0.009,Y -287.571,Z 965.678,A 0.000,B 0.000,C 90.000,E1 302.005} C_DIS
LIN {X -0.042,Y -307.307,Z 965.661,A 0.000,B 0.000,C 90.000,E1 298.999} C_DIS
LIN {X -0.066,Y -321.804,Z 965.650,A 0.000,B 0.000,C 90.000,E1 297.052} C_DIS
LIN {X 0.027,Y -337.602,Z 965.640,A 0.000,B 0.000,C 90.000,E1 295.155} C_DIS
LIN {X -0.053,Y -361.848,Z 965.625,A 0.000,B 0.000,C 90.000,E1 292.589} C_DIS
LIN {X -0.157,Y -380.500,Z 965.615,A 0.000,B 0.000,C 90.000,E1 290.737} C_DIS
LIN {X 0.017,Y -396.619,Z 965.606,A 0.000,B 0.000,C 90.000,E1 289.141} C_DIS
LIN {X 0.046,Y -404.463,Z 965.602,A 0.000,B 0.000,C 90.000,E1 288.362} C_DIS
LIN {X -0.104,Y -414.662,Z 965.596,A 0.000,B 0.000,C 90.000,E1 287.330} C_DIS
LIN {X -0.142,Y -424.604,Z 965.590,A 0.000,B 0.000,C 90.000,E1 286.260} C_DIS
LIN {X -0.222,Y -434.051,Z 965.584,A 0.000,B 0.000,C 90.000,E1 285.190} C_DIS
LIN {X -0.191,Y -442.852,Z 965.578,A 0.000,B 0.000,C 90.000,E1 284.120} C_DIS
LIN {X -0.162,Y -451.187,Z 965.572,A 0.000,B 0.000,C 90.000,E1 283.063} C_DIS
LIN {X -0.204,Y -461.017,Z 965.565,A 0.000,B 0.000,C 90.000,E1 281.771} C_DIS
LIN {X 0.042,Y -468.475,Z 965.560,A 0.000,B 0.000,C 90.000,E1 280.715} C_DIS
LIN {X -0.035,Y -473.644,Z 965.555,A 0.000,B 0.000,C 90.000,E1 279.962} C_DIS
LIN {X -0.058,Y -478.122,Z 965.551,A 0.000,B 0.000,C 90.000,E1 279.208} C_DIS
LIN {X -0.044,Y -482.002,Z 965.547,A 0.000,B 0.000,C 90.000,E1 278.454} C_DIS
LIN {X 0.123,Y -484.231,Z 965.544,A 0.000,B 0.000,C 90.000,E1 277.936} C_DIS
LIN {X -0.113,Y -486.157,Z 965.541,A 0.000,B 0.000,C 90.000,E1 277.466} C_DIS
LIN {X 0.074,Y -487.786,Z 965.539,A 0.000,B 0.000,C 90.000,E1 276.947} C_DIS
LIN {X -0.212,Y -489.067,Z 965.536,A 0.000,B 0.000,C 90.000,E1 276.486} C_DIS
LIN {X -0.003,Y -489.998,Z 965.533,A 0.000,B 0.000,C 90.000,E1 275.967} C_DIS
LIN {X 0.165,Y -490.594,Z 965.530,A 0.000,B 0.000,C 90.000,E1 275.454} C_DIS
LIN {X -0.099,Y -490.899,Z 965.528,A 0.000,B 0.000,C 90.000,E1 274.992} C_DIS
LIN {X 0.126,Y -490.745,Z 965.525,A 0.000,B 0.000,C 90.000,E1 274.473} C_DIS
LIN {X -0.138,Y -490.116,Z 965.522,A 0.000,B 0.000,C 90.000,E1 274.012} C_DIS
LIN {X 0.052,Y -488.981,Z 965.519,A 0.000,B 0.000,C 90.000,E1 273.498} C_DIS
LIN {X -0.219,Y -487.326,Z 965.517,A 0.000,B 0.000,C 90.000,E1 273.037} C_DIS
LIN {X -0.036,Y -484.979,Z 965.514,A 0.000,B 0.000,C 90.000,E1 272.522} C_DIS
LIN {X 0.134,Y -481.938,Z 965.511,A 0.000,B 0.000,C 90.000,E1 272.007} C_DIS
LIN {X -0.176,Y -478.003,Z 965.508,A 0.000,B 0.000,C 90.000,E1 271.547} C_DIS
LIN {X 0.128,Y -475.688,Z 965.507,A 0.000,B 0.000,C 90.000,E1 271.260} C_DIS
LIN {X -0.128,Y -470.279,Z 965.504,A 0.000,B 0.000,C 90.000,E1 270.802} C_DIS
LIN {X -0.077,Y -464.370,Z 965.502,A 0.000,B 0.000,C 90.000,E1 270.344} C_DIS
LIN {X -0.062,Y -458.075,Z 965.500,A 0.000,B 0.000,C 90.000,E1 269.943} C_DIS
LIN {X -0.099,Y -451.421,Z 965.498,A 0.000,B 0.000,C 90.000,E1 269.599} C_DIS
LIN {X -0.169,Y -444.419,Z 965.496,A 0.000,B 0.000,C 90.000,E1 269.312} C_DIS
LIN {X 0.144,Y -437.199,Z 965.495,A 0.000,B 0.000,C 90.000,E1 269.026} C_DIS
LIN {X -0.073,Y -429.414,Z 965.494,A 0.000,B 0.000,C 90.000,E1 268.854} C_DIS
LIN {X 0.036,Y -421.641,Z 965.493,A 0.000,B 0.000,C 90.000,E1 268.682} C_DIS
LIN {X -0.010,Y -413.162,Z 965.492,A 0.000,B 0.000,C 90.000,E1 268.568} C_DIS
LIN {X 0.025,Y -406.028,Z 965.492,A 0.000,B 0.000,C 90.000,E1 268.511} C_DIS
LIN {X -0.086,Y -400.004,Z 965.492,A 0.000,B 0.000,C 90.000,E1 268.511} C_DIS
LIN {X -0.064,Y -181.212,Z 965.492,A 0.000,B 0.000,C 90.000,E1 268.511} C_DIS
LIN {X 0.048,Y -180.878,Z 965.473,A 0.000,B 0.000,C 90.000,E1 265.065} C_DIS
LIN {X -0.072,Y -178.996,Z 965.445,A 0.000,B 0.000,C 90.000,E1 260.038} C_DIS
LIN {X 0.022,Y -178.584,Z 965.440,A 0.000,B 0.000,C 90.000,E1 259.162} C_DIS
LIN {X -0.084,Y -175.637,Z 965.411,A 0.000,B 0.000,C 90.000,E1 254.102} C_DIS
LIN {X -0.018,Y -172.357,Z 965.388,A 0.000,B 0.000,C 90.000,E1 249.806} C_DIS
LIN {X -0.063,Y -171.141,Z 965.378,A 0.000,B 0.000,C 90.000,E1 248.103} C_DIS
LIN {X -0.019,Y -167.445,Z 965.354,A 0.000,B 0.000,C 90.000,E1 243.768} C_DIS
LIN {X 0.064,Y -166.841,Z 965.349,A 0.000,B 0.000,C 90.000,E1 242.871} C_DIS
LIN {X -0.019,Y -162.825,Z 965.325,A 0.000,B 0.000,C 90.000,E1 238.535} C_DIS
LIN {X 0.044,Y -161.510,Z 965.315,A 0.000,B 0.000,C 90.000,E1 236.755} C_DIS
LIN {X -0.003,Y -157.508,Z 965.291,A 0.000,B 0.000,C 90.000,E1 232.351} C_DIS
LIN {X 0.031,Y -155.530,Z 965.276,A 0.000,B 0.000,C 90.000,E1 229.666} C_DIS
LIN {X 0.080,Y -151.827,Z 965.251,A 0.000,B 0.000,C 90.000,E1 225.162} C_DIS
LIN {X -0.009,Y -150.042,Z 965.236,A 0.000,B 0.000,C 90.000,E1 222.486} C_DIS
LIN {X 0.006,Y -146.858,Z 965.211,A 0.000,B 0.000,C 90.000,E1 217.935} C_DIS
LIN {X 0.024,Y -145.442,Z 965.195,A 0.000,B 0.000,C 90.000,E1 215.185} C_DIS
LIN {X 0.019,Y -142.862,Z 965.170,A 0.000,B 0.000,C 90.000,E1 210.590} C_DIS
LIN {X 0.072,Y -141.478,Z 965.149,A 0.000,B 0.000,C 90.000,E1 206.873} C_DIS
LIN {X -0.069,Y -139.381,Z 965.113,A 0.000,B 0.000,C 90.000,E1 200.429} C_DIS
LIN {X 0.052,Y -138.834,Z 965.098,A 0.000,B 0.000,C 90.000,E1 197.583} C_DIS
LIN {X -0.020,Y -138.354,Z 965.056,A 0.000,B 0.000,C 90.000,E1 190.141} C_DIS
LIN {X -0.025,Y -139.524,Z 965.004,A 0.000,B 0.000,C 90.000,E1 180.802} C_DIS
LIN {X 0.056,Y -141.193,Z 964.973,A 0.000,B 0.000,C 90.000,E1 175.184} C_DIS
LIN {X 0.027,Y -142.570,Z 964.958,A 0.000,B 0.000,C 90.000,E1 172.413} C_DIS
LIN {X -0.018,Y -144.857,Z 964.932,A 0.000,B 0.000,C 90.000,E1 167.813} C_DIS
LIN {X -0.063,Y -147.483,Z 964.912,A 0.000,B 0.000,C 90.000,E1 164.157} C_DIS
LIN {X -0.037,Y -150.069,Z 964.892,A 0.000,B 0.000,C 90.000,E1 160.496} C_DIS
LIN {X -0.033,Y -153.418,Z 964.871,A 0.000,B 0.000,C 90.000,E1 156.869} C_DIS
LIN {X 0.016,Y -156.838,Z 964.851,A 0.000,B 0.000,C 90.000,E1 153.256} C_DIS
LIN {X 0.087,Y -160.918,Z 964.832,A 0.000,B 0.000,C 90.000,E1 149.665} C_DIS
LIN {X 0.032,Y -163.042,Z 964.822,A 0.000,B 0.000,C 90.000,E1 147.916} C_DIS
LIN {X 0.036,Y -167.434,Z 964.802,A 0.000,B 0.000,C 90.000,E1 144.402} C_DIS
LIN {X -0.055,Y -171.272,Z 964.788,A 0.000,B 0.000,C 90.000,E1 141.823} C_DIS
LIN {X -0.015,Y -176.165,Z 964.769,A 0.000,B 0.000,C 90.000,E1 138.366} C_DIS
LIN {X -0.018,Y -180.436,Z 964.754,A 0.000,B 0.000,C 90.000,E1 135.810} C_DIS
LIN {X -0.042,Y -185.841,Z 964.736,A 0.000,B 0.000,C 90.000,E1 132.447} C_DIS
LIN {X 0.012,Y -190.464,Z 964.722,A 0.000,B 0.000,C 90.000,E1 129.930} C_DIS
LIN {X -0.025,Y -194.976,Z 964.707,A 0.000,B 0.000,C 90.000,E1 127.317} C_DIS
LIN {X -0.074,Y -298.348,Z 964.707,A 0.000,B 0.000,C 90.000,E1 127.317} C_DIS
LIN {X 0.109,Y -300.588,Z 964.707,A 0.000,B 0.000,C 90.000,E1 127.237} C_DIS
LIN {X -0.010,Y -305.915,Z 964.705,A 0.000,B 0.000,C 90.000,E1 126.950} C_DIS
LIN {X -0.132,Y -308.813,Z 964.704,A 0.000,B 0.000,C 90.000,E1 126.664} C_DIS
LIN {X -0.186,Y -310.837,Z 964.702,A 0.000,B 0.000,C 90.000,E1 126.377} C_DIS
LIN {X 0.197,Y -312.423,Z 964.700,A 0.000,B 0.000,C 90.000,E1 126.011} C_DIS
LIN {X -0.012,Y -313.802,Z 964.698,A 0.000,B 0.000,C 90.000,E1 125.724} C_DIS
LIN {X -0.019,Y -326.625,Z 964.677,A 0.000,B 0.000,C 90.000,E1 121.878} C_DIS
LIN {X -0.172,Y -337.664,Z 964.661,A 0.000,B 0.000,C 90.000,E1 119.077} C_DIS
LIN {X -0.048,Y -350.096,Z 964.646,A 0.000,B 0.000,C 90.000,E1 116.283} C_DIS
LIN {X -0.038,Y -364.037,Z 964.631,A 0.000,B 0.000,C 90.000,E1 113.567} C_DIS
LIN {X -0.168,Y -377.793,Z 964.618,A 0.000,B 0.000,C 90.000,E1 111.227} C_DIS
LIN {X -0.085,Y -392.934,Z 964.605,A 0.000,B 0.000,C 90.000,E1 108.906} C_DIS
LIN {X 0.133,Y -409.568,Z 964.592,A 0.000,B 0.000,C 90.000,E1 106.622} C_DIS
LIN {X 0.152,Y -427.816,Z 964.580,A 0.000,B 0.000,C 90.000,E1 104.426} C_DIS
LIN {X -0.146,Y -447.554,Z 964.569,A 0.000,B 0.000,C 90.000,E1 102.355} C_DIS
LIN {X 0.228,Y -467.829,Z 964.558,A 0.000,B 0.000,C 90.000,E1 100.366} C_DIS
LIN {X 0.113,Y -469.782,Z 964.556,A 0.000,B 0.000,C 90.000,E1 100.141} C_DIS
LIN {X 0.081,Y -471.265,Z 964.555,A 0.000,B 0.000,C 90.000,E1 99.905} C_DIS
LIN {X -0.065,Y -472.449,Z 964.554,A 0.000,B 0.000,C 90.000,E1 99.670} C_DIS
LIN {X 0.255,Y -473.312,Z 964.552,A 0.000,B 0.000,C 90.000,E1 99.378} C_DIS
LIN {X -0.101,Y -474.221,Z 964.549,A 0.000,B 0.000,C 90.000,E1 98.916} C_DIS
LIN {X 0.018,Y -474.152,Z 964.547,A 0.000,B 0.000,C 90.000,E1 98.398} C_DIS
LIN {X 0.210,Y -473.102,Z 964.544,A 0.000,B 0.000,C 90.000,E1 97.871} C_DIS
LIN {X 0.006,Y -472.161,Z 964.542,A 0.000,B 0.000,C 90.000,E1 97.644} C_DIS
LIN {X -0.134,Y -470.887,Z 964.541,A 0.000,B 0.000,C 90.000,E1 97.409} C_DIS
LIN {X -0.072,Y -459.165,Z 964.531,A 0.000,B 0.000,C 90.000,E1 95.625} C_DIS
LIN {X 0.213,Y -447.389,Z 964.521,A 0.000,B 0.000,C 90.000,E1 93.784} C_DIS
LIN {X -0.063,Y -433.963,Z 964.510,A 0.000,B 0.000,C 90.000,E1 91.718} C_DIS
LIN {X 0.109,Y -416.742,Z 964.493,A 0.000,B 0.000,C 90.000,E1 88.740} C_DIS
LIN {X -0.070,Y -406.222,Z 964.482,A 0.000,B 0.000,C 90.000,E1 86.846} C_DIS
LIN {X -0.060,Y -395.512,Z 964.472,A 0.000,B 0.000,C 90.000,E1 84.894} C_DIS
LIN {X 0.188,Y -384.693,Z 964.461,A 0.000,B 0.000,C 90.000,E1 82.875} C_DIS
LIN {X -0.152,Y -376.807,Z 964.453,A 0.000,B 0.000,C 90.000,E1 81.489} C_DIS
LIN {X 0.167,Y -365.343,Z 964.441,A 0.000,B 0.000,C 90.000,E1 79.398} C_DIS
LIN {X 0.030,Y -357.027,Z 964.433,A 0.000,B 0.000,C 90.000,E1 77.937} C_DIS
LIN {X 0.058,Y -343.541,Z 964.420,A 0.000,B 0.000,C 90.000,E1 75.519} C_DIS
LIN {X -0.023,Y -326.228,Z 964.401,A 0.000,B 0.000,C 90.000,E1 72.127} C_DIS
LIN {X 0.123,Y -315.609,Z 964.388,A 0.000,B 0.000,C 90.000,E1 69.880} C_DIS
LIN {X 0.046,Y -303.574,Z 964.374,A 0.000,B 0.000,C 90.000,E1 67.305} C_DIS
LIN {X 0.025,Y -291.690,Z 964.359,A 0.000,B 0.000,C 90.000,E1 64.665} C_DIS
LIN {X 0.136,Y -281.399,Z 964.346,A 0.000,B 0.000,C 90.000,E1 62.281} C_DIS
LIN {X -0.088,Y -271.160,Z 964.333,A 0.000,B 0.000,C 90.000,E1 59.921} C_DIS
LIN {X -0.116,Y -259.859,Z 964.317,A 0.000,B 0.000,C 90.000,E1 57.120} C_DIS
LIN {X -0.001,Y -247.684,Z 964.299,A 0.000,B 0.000,C 90.000,E1 53.863} C_DIS
LIN {X -0.034,Y -236.383,Z 964.281,A 0.000,B 0.000,C 90.000,E1 50.561} C_DIS
LIN {X 0.082,Y -225.939,Z 964.262,A 0.000,B 0.000,C 90.000,E1 47.148} C_DIS
LIN {X -0.028,Y -217.260,Z 964.245,A 0.000,B 0.000,C 90.000,E1 44.109} C_DIS
LIN {X -0.015,Y -209.071,Z 964.228,A 0.000,B 0.000,C 90.000,E1 40.987} C_DIS
LIN {X -0.002,Y -201.499,Z 964.210,A 0.000,B 0.000,C 90.000,E1 37.810} C_DIS
LIN {X -0.096,Y -194.559,Z 964.192,A 0.000,B 0.000,C 90.000,E1 34.612} C_DIS
LIN {X -0.094,Y -188.295,Z 964.174,A 0.000,B 0.000,C 90.000,E1 31.337} C_DIS
LIN {X 0.042,Y -182.747,Z 964.156,A 0.000,B 0.000,C 90.000,E1 27.975} C_DIS
LIN {X -0.056,Y -177.885,Z 964.137,A 0.000,B 0.000,C 90.000,E1 24.643} C_DIS
LIN {X -0.004,Y -173.754,Z 964.118,A 0.000,B 0.000,C 90.000,E1 21.227} C_DIS
LIN {X -0.075,Y -170.319,Z 964.099,A 0.000,B 0.000,C 90.000,E1 17.819} C_DIS
LIN {X 0.000,Y -166.982,Z 964.075,A 0.000,B 0.000,C 90.000,E1 13.467} C_DIS
LIN {X 0.038,Y -164.321,Z 964.046,A 0.000,B 0.000,C 90.000,E1 8.219} C_DIS
LIN {X -0.047,Y -165.254,Z 963.958,A 0.000,B 0.000,C 90.000,E1 352.527} C_DIS
LIN {X -0.089,Y -167.864,Z 963.934,A 0.000,B 0.000,C 90.000,E1 348.173} C_DIS
LIN {X -0.044,Y -170.789,Z 963.915,A 0.000,B 0.000,C 90.000,E1 344.685} C_DIS
LIN {X -0.017,Y -175.422,Z 963.891,A 0.000,B 0.000,C 90.000,E1 340.369} C_DIS
LIN {X -0.067,Y -179.987,Z 963.872,A 0.000,B 0.000,C 90.000,E1 336.975} C_DIS
LIN {X -0.030,Y -185.307,Z 963.853,A 0.000,B 0.000,C 90.000,E1 333.589} C_DIS
LIN {X -0.027,Y -191.286,Z 963.835,A 0.000,B 0.000,C 90.000,E1 330.255} C_DIS
LIN {X -0.007,Y -197.942,Z 963.816,A 0.000,B 0.000,C 90.000,E1 326.962} C_DIS
LIN {X 0.065,Y -205.098,Z 963.798,A 0.000,B 0.000,C 90.000,E1 323.703} C_DIS
LIN {X -0.038,Y -213.852,Z 963.779,A 0.000,B 0.000,C 90.000,E1 320.150} C_DIS
LIN {X -0.022,Y -222.274,Z 963.761,A 0.000,B 0.000,C 90.000,E1 317.025} C_DIS
LIN {X 0.035,Y -231.610,Z 963.744,A 0.000,B 0.000,C 90.000,E1 313.947} C_DIS
LIN {X 0.085,Y -239.521,Z 963.732,A 0.000,B 0.000,C 90.000,E1 311.676} C_DIS
LIN {X -0.038,Y -249.912,Z 963.717,A 0.000,B 0.000,C 90.000,E1 309.116} C_DIS
LIN {X 0.045,Y -258.305,Z 963.707,A 0.000,B 0.000,C 90.000,E1 307.282} C_DIS
LIN {X -0.010,Y -273.356,Z 963.691,A 0.000,B 0.000,C 90.000,E1 304.452} C_DIS
LIN {X 0.069,Y -291.820,Z 963.674,A 0.000,B 0.000,C 90.000,E1 301.337} C_DIS
LIN {X -0.041,Y -309.618,Z 963.659,A 0.000,B 0.000,C 90.000,E1 298.693} C_DIS
LIN {X -0.014,Y -324.266,Z 963.649,A 0.000,B 0.000,C 90.000,E1 296.744} C_DIS
LIN {X 0.183,Y -348.336,Z 963.633,A 0.000,B 0.000,C 90.000,E1 293.951} C_DIS
LIN {X 0.098,Y -367.111,Z 963.622,A 0.000,B 0.000,C 90.000,E1 292.025} C_DIS
LIN {X 0.047,Y -383.226,Z 963.614,A 0.000,B 0.000,C 90.000,E1 290.429} C_DIS
LIN {X -0.043,Y -396.564,Z 963.606,A 0.000,B 0.000,C 90.000,E1 289.141} C_DIS
LIN {X -0.089,Y -406.964,Z 963.601,A 0.000,B 0.000,C 90.000,E1 288.109} C_DIS
LIN {X -0.027,Y -417.132,Z 963.595,A 0.000,B 0.000,C 90.000,E1 287.040} C_DIS
LIN {X -0.108,Y -426.996,Z 963.589,A 0.000,B 0.000,C 90.000,E1 285.969} C_DIS
LIN {X -0.156,Y -436.250,Z 963.583,A 0.000,B 0.000,C 90.000,E1 284.898} C_DIS
LIN {X -0.096,Y -444.889,Z 963.577,A 0.000,B 0.000,C 90.000,E1 283.828} C_DIS
LIN {X -0.039,Y -453.097,Z 963.571,A 0.000,B 0.000,C 90.000,E1 282.771} C_DIS
LIN {X -0.056,Y -462.888,Z 963.564,A 0.000,B 0.000,C 90.000,E1 281.478} C_DIS
LIN {X 0.130,Y -470.263,Z 963.558,A 0.000,B 0.000,C 90.000,E1 280.433} C_DIS
LIN {X 0.161,Y -475.209,Z 963.554,A 0.000,B 0.000,C 90.000,E1 279.670} C_DIS
LIN {X 0.148,Y -479.523,Z 963.550,A 0.000,B 0.000,C 90.000,E1 278.916} C_DIS
LIN {X 0.178,Y -483.184,Z 963.545,A 0.000,B 0.000,C 90.000,E1 278.163} C_DIS
LIN {X 0.234,Y -486.210,Z 963.541,A 0.000,B 0.000,C 90.000,E1 277.409} C_DIS
LIN {X -0.061,Y -487.842,Z 963.539,A 0.000,B 0.000,C 90.000,E1 276.947} C_DIS
LIN {X 0.138,Y -489.111,Z 963.536,A 0.000,B 0.000,C 90.000,E1 276.429} C_DIS
LIN {X -0.138,Y -490.057,Z 963.533,A 0.000,B 0.000,C 90.000,E1 275.967} C_DIS
LIN {X 0.030,Y -490.670,Z 963.530,A 0.000,B 0.000,C 90.000,E1 275.454} C_DIS
LIN {X -0.234,Y -490.941,Z 963.528,A 0.000,B 0.000,C 90.000,E1 274.992} C_DIS
LIN {X -0.008,Y -490.788,Z 963.525,A 0.000,B 0.000,C 90.000,E1 274.473} C_DIS
LIN {X 0.217,Y -490.150,Z 963.522,A 0.000,B 0.000,C 90.000,E1 273.955} C_DIS
LIN {X -0.082,Y -489.022,Z 963.519,A 0.000,B 0.000,C 90.000,E1 273.498} C_DIS
LIN {X 0.135,Y -487.351,Z 963.517,A 0.000,B 0.000,C 90.000,E1 272.980} C_DIS
LIN {X -0.168,Y -485.041,Z 963.514,A 0.000,B 0.000,C 90.000,E1 272.522} C_DIS
LIN {X 0.004,Y -481.940,Z 963.511,A 0.000,B 0.000,C 90.000,E1 272.007} C_DIS
LIN {X 0.171,Y -478.007,Z 963.508,A 0.000,B 0.000,C 90.000,E1 271.489} C_DIS
LIN {X -0.171,Y -473.059,Z 963.506,A 0.000,B 0.000,C 90.000,E1 271.031} C_DIS
LIN {X 0.129,Y -467.251,Z 963.503,A 0.000,B 0.000,C 90.000,E1 270.516} C_DIS
LIN {X -0.064,Y -461.139,Z 963.501,A 0.000,B 0.000,C 90.000,E1 270.115} C_DIS
LIN {X 0.156,Y -454.681,Z 963.499,A 0.000,B 0.000,C 90.000,E1 269.714} C_DIS
LIN {X -0.152,Y -447.682,Z 963.497,A 0.000,B 0.000,C 90.000,E1 269.427} C_DIS
LIN {X -0.004,Y -440.693,Z 963.495,A 0.000,B 0.000,C 90.000,E1 269.141} C_DIS
LIN {X 0.056,Y -433.343,Z 963.494,A 0.000,B 0.000,C 90.000,E1 268.912} C_DIS
LIN {X 0.008,Y -425.434,Z 963.493,A 0.000,B 0.000,C 90.000,E1 268.740} C_DIS
LIN {X -0.168,Y -417.435,Z 963.492,A 0.000,B 0.000,C 90.000,E1 268.625} C_DIS
LIN {X -0.101,Y -406.255,Z 963.492,A 0.000,B 0.000,C 90.000,E1 268.511} C_DIS
LIN {X -0.158,Y -404.021,Z 963.492,A 0.000,B 0.000,C 90.000,E1 268.511} C_DIS
LIN {X 0.084,Y -181.210,Z 963.492,A 0.000,B 0.000,C 90.000,E1 268.453} C_DIS
LIN {X -0.015,Y -180.875,Z 963.473,A 0.000,B 0.000,C 90.000,E1 265.065} C_DIS
LIN {X 0.041,Y -178.992,Z 963.444,A 0.000,B 0.000,C 90.000,E1 259.982} C_DIS
LIN {X 0.052,Y -177.978,Z 963.435,A 0.000,B 0.000,C 90.000,E1 258.285} C_DIS
LIN {X 0.022,Y -175.623,Z 963.411,A 0.000,B 0.000,C 90.000,E1 254.047} C_DIS
LIN {X 0.082,Y -172.343,Z 963.388,A 0.000,B 0.000,C 90.000,E1 249.752} C_DIS
LIN {X 0.061,Y -171.819,Z 963.383,A 0.000,B 0.000,C 90.000,E1 248.901} C_DIS
LIN {X 0.068,Y -170.287,Z 963.373,A 0.000,B 0.000,C 90.000,E1 247.177} C_DIS
LIN {X 0.004,Y -166.826,Z 963.349,A 0.000,B 0.000,C 90.000,E1 242.871} C_DIS
LIN {X -0.079,Y -162.808,Z 963.325,A 0.000,B 0.000,C 90.000,E1 238.535} C_DIS
LIN {X -0.015,Y -161.495,Z 963.315,A 0.000,B 0.000,C 90.000,E1 236.755} C_DIS
LIN {X -0.061,Y -157.492,Z 963.291,A 0.000,B 0.000,C 90.000,E1 232.351} C_DIS
LIN {X -0.027,Y -155.510,Z 963.276,A 0.000,B 0.000,C 90.000,E1 229.666} C_DIS
LIN {X 0.023,Y -151.812,Z 963.251,A 0.000,B 0.000,C 90.000,E1 225.162} C_DIS
LIN {X 0.036,Y -150.025,Z 963.236,A 0.000,B 0.000,C 90.000,E1 222.447} C_DIS
LIN {X -0.050,Y -146.845,Z 963.211,A 0.000,B 0.000,C 90.000,E1 217.935} C_DIS
LIN {X -0.031,Y -145.428,Z 963.195,A 0.000,B 0.000,C 90.000,E1 215.185} C_DIS
LIN {X -0.035,Y -142.852,Z 963.170,A 0.000,B 0.000,C 90.000,E1 210.590} C_DIS
LIN {X 0.017,Y -141.468,Z 963.149,A 0.000,B 0.000,C 90.000,E1 206.873} C_DIS
LIN {X 0.008,Y -139.377,Z 963.113,A 0.000,B 0.000,C 90.000,E1 200.375} C_DIS
LIN {X -0.002,Y -138.829,Z 963.098,A 0.000,B 0.000,C 90.000,E1 197.583} C_DIS
LIN {X -0.074,Y -138.353,Z 963.056,A 0.000,B 0.000,C 90.000,E1 190.141} C_DIS
LIN {X 0.060,Y -139.528,Z 963.004,A 0.000,B 0.000,C 90.000,E1 180.745} C_DIS
LIN {X 0.014,Y -141.202,Z 962.973,A 0.000,B 0.000,C 90.000,E1 175.179} C_DIS
LIN {X -0.027,Y -142.578,Z 962.958,A 0.000,B 0.000,C 90.000,E1 172.413} C_DIS
LIN {X 0.068,Y -144.870,Z 962.932,A 0.000,B 0.000,C 90.000,E1 167.757} C_DIS
LIN {X 0.023,Y -147.498,Z 962.912,A 0.000,B 0.000,C 90.000,E1 164.102} C_DIS
LIN {X -0.043,Y -150.087,Z 962.891,A 0.000,B 0.000,C 90.000,E1 160.477} C_DIS
LIN {X -0.030,Y -153.439,Z 962.871,A 0.000,B 0.000,C 90.000,E1 156.847} C_DIS
LIN {X -0.036,Y -157.803,Z 962.846,A 0.000,B 0.000,C 90.000,E1 152.359} C_DIS
LIN {X -0.004,Y -162.084,Z 962.827,A 0.000,B 0.000,C 90.000,E1 148.791} C_DIS
LIN {X 0.021,Y -166.283,Z 962.807,A 0.000,B 0.000,C 90.000,E1 145.261} C_DIS
LIN {X 0.018,Y -171.300,Z 962.788,A 0.000,B 0.000,C 90.000,E1 141.778} C_DIS
LIN {X 0.054,Y -176.197,Z 962.769,A 0.000,B 0.000,C 90.000,E1 138.324} C_DIS
LIN {X -0.081,Y -180.471,Z 962.754,A 0.000,B 0.000,C 90.000,E1 135.810} C_DIS
LIN {X 0.030,Y -185.876,Z 962.736,A 0.000,B 0.000,C 90.000,E1 132.405} C_DIS
LIN {X -0.054,Y -190.501,Z 962.722,A 0.000,B 0.000,C 90.000,E1 129.930} C_DIS
LIN {X -0.064,Y -194.913,Z 962.707,A 0.000,B 0.000,C 90.000,E1 127.363} C_DIS
LIN {X 0.088,Y -298.235,Z 962.707,A 0.000,B 0.000,C 90.000,E1 127.317} C_DIS
LIN {X -0.069,Y -299.920,Z 962.707,A 0.000,B 0.000,C 90.000,E1 127.317} C_DIS
LIN {X -0.124,Y -303.759,Z 962.706,A 0.000,B 0.000,C 90.000,E1 127.156} C_DIS
LIN {X 0.062,Y -305.991,Z 962.705,A 0.000,B 0.000,C 90.000,E1 126.950} C_DIS
LIN {X -0.052,Y -309.079,Z 962.703,A 0.000,B 0.000,C 90.000,E1 126.629} C_DIS
LIN {X 0.098,Y -311.066,Z 962.702,A 0.000,B 0.000,C 90.000,E1 126.297} C_DIS
LIN {X -0.002,Y -312.622,Z 962.700,A 0.000,B 0.000,C 90.000,E1 126.011} C_DIS
LIN {X 0.046,Y -313.934,Z 962.698,A 0.000,B 0.000,C 90.000,E1 125.678} C_DIS
LIN {X 0.132,Y -325.588,Z 962.679,A 0.000,B 0.000,C 90.000,E1 122.133} C_DIS
LIN {X -0.049,Y -336.491,Z 962.663,A 0.000,B 0.000,C 90.000,E1 119.333} C_DIS
LIN {X 0.040,Y -348.783,Z 962.647,A 0.000,B 0.000,C 90.000,E1 116.539} C_DIS
LIN {X 0.022,Y -362.567,Z 962.632,A 0.000,B 0.000,C 90.000,E1 113.823} C_DIS
LIN {X -0.001,Y -376.174,Z 962.619,A 0.000,B 0.000,C 90.000,E1 111.461} C_DIS
LIN {X 0.040,Y -391.155,Z 962.606,A 0.000,B 0.000,C 90.000,E1 109.141} C_DIS
LIN {X -0.177,Y -407.617,Z 962.594,A 0.000,B 0.000,C 90.000,E1 106.913} C_DIS
LIN {X -0.227,Y -425.679,Z 962.582,A 0.000,B 0.000,C 90.000,E1 104.717} C_DIS
LIN {X -0.217,Y -445.288,Z 962.570,A 0.000,B 0.000,C 90.000,E1 102.591} C_DIS
LIN {X 0.010,Y -468.052,Z 962.558,A 0.000,B 0.000,C 90.000,E1 100.366} C_DIS
LIN {X -0.125,Y -469.966,Z 962.556,A 0.000,B 0.000,C 90.000,E1 100.141} C_DIS
LIN {X -0.178,Y -471.419,Z 962.555,A 0.000,B 0.000,C 90.000,E1 99.905} C_DIS
LIN {X -0.004,Y -473.394,Z 962.552,A 0.000,B 0.000,C 90.000,E1 99.378} C_DIS
LIN {X 0.102,Y -474.246,Z 962.549,A 0.000,B 0.000,C 90.000,E1 98.859} C_DIS
LIN {X -0.246,Y -474.123,Z 962.547,A 0.000,B 0.000,C 90.000,E1 98.398} C_DIS
LIN {X -0.054,Y -473.013,Z 962.544,A 0.000,B 0.000,C 90.000,E1 97.871} C_DIS
LIN {X 0.211,Y -472.036,Z 962.542,A 0.000,B 0.000,C 90.000,E1 97.587} C_DIS
LIN {X 0.070,Y -470.720,Z 962.541,A 0.000,B 0.000,C 90.000,E1 97.352} C_DIS
LIN {X 0.125,Y -458.986,Z 962.531,A 0.000,B 0.000,C 90.000,E1 95.568} C_DIS
LIN {X -0.044,Y -447.255,Z 962.521,A 0.000,B 0.000,C 90.000,E1 93.784} C_DIS
LIN {X 0.119,Y -433.853,Z 962.509,A 0.000,B 0.000,C 90.000,E1 91.661} C_DIS
LIN {X 0.177,Y -418.124,Z 962.494,A 0.000,B 0.000,C 90.000,E1 88.969} C_DIS
LIN {X -0.001,Y -407.609,Z 962.484,A 0.000,B 0.000,C 90.000,E1 87.078} C_DIS
LIN {X 0.065,Y -396.899,Z 962.473,A 0.000,B 0.000,C 90.000,E1 85.122} C_DIS
LIN {X -0.091,Y -386.099,Z 962.462,A 0.000,B 0.000,C 90.000,E1 83.166} C_DIS
LIN {X -0.029,Y -378.243,Z 962.454,A 0.000,B 0.000,C 90.000,E1 81.724} C_DIS
LIN {X -0.041,Y -368.469,Z 962.444,A 0.000,B 0.000,C 90.000,E1 79.982} C_DIS
LIN {X -0.158,Y -358.537,Z 962.434,A 0.000,B 0.000,C 90.000,E1 78.229} C_DIS
LIN {X -0.099,Y -346.710,Z 962.423,A 0.000,B 0.000,C 90.000,E1 76.117} C_DIS
LIN {X 0.048,Y -330.654,Z 962.406,A 0.000,B 0.000,C 90.000,E1 73.015} C_DIS
LIN {X 0.196,Y -319.978,Z 962.393,A 0.000,B 0.000,C 90.000,E1 70.786} C_DIS
LIN {X -0.089,Y -309.402,Z 962.381,A 0.000,B 0.000,C 90.000,E1 68.592} C_DIS
LIN {X 0.028,Y -300.414,Z 962.370,A 0.000,B 0.000,C 90.000,E1 66.613} C_DIS
LIN {X 0.075,Y -290.060,Z 962.357,A 0.000,B 0.000,C 90.000,E1 64.280} C_DIS
LIN {X 0.145,Y -279.751,Z 962.344,A 0.000,B 0.000,C 90.000,E1 61.897} C_DIS
LIN {X -0.112,Y -269.531,Z 962.331,A 0.000,B 0.000,C 90.000,E1 59.537} C_DIS
LIN {X 0.051,Y -259.673,Z 962.317,A 0.000,B 0.000,C 90.000,E1 57.041} C_DIS
LIN {X -0.043,Y -247.493,Z 962.299,A 0.000,B 0.000,C 90.000,E1 53.829} C_DIS
LIN {X -0.037,Y -236.259,Z 962.281,A 0.000,B 0.000,C 90.000,E1 50.517} C_DIS
LIN {X -0.098,Y -225.835,Z 962.262,A 0.000,B 0.000,C 90.000,E1 47.148} C_DIS
LIN {X 0.110,Y -217.188,Z 962.245,A 0.000,B 0.000,C 90.000,E1 44.028} C_DIS
LIN {X -0.021,Y -209.035,Z 962.227,A 0.000,B 0.000,C 90.000,E1 40.943} C_DIS
LIN {X 0.121,Y -201.479,Z 962.210,A 0.000,B 0.000,C 90.000,E1 37.729} C_DIS
LIN {X 0.020,Y -194.576,Z 962.192,A 0.000,B 0.000,C 90.000,E1 34.532} C_DIS
LIN {X 0.016,Y -188.334,Z 962.174,A 0.000,B 0.000,C 90.000,E1 31.258} C_DIS
LIN {X -0.102,Y -182.813,Z 962.155,A 0.000,B 0.000,C 90.000,E1 27.975} C_DIS
LIN {X -0.031,Y -177.954,Z 962.137,A 0.000,B 0.000,C 90.000,E1 24.591} C_DIS
LIN {X 0.026,Y -173.828,Z 962.118,A 0.000,B 0.000,C 90.000,E1 21.173} C_DIS
LIN {X -0.041,Y -170.397,Z 962.099,A 0.000,B 0.000,C 90.000,E1 17.764} C_DIS
LIN {X 0.038,Y -167.079,Z 962.075,A 0.000,B 0.000,C 90.000,E1 13.411} C_DIS
LIN {X 0.083,Y -164.446,Z 962.046,A 0.000,B 0.000,C 90.000,E1 8.163} C_DIS
LIN {X -0.016,Y -165.042,Z 961.963,A 0.000,B 0.000,C 90.000,E1 353.394} C_DIS
LIN {X -0.075,Y -168.056,Z 961.934,A 0.000,B 0.000,C 90.000,E1 348.173} C_DIS
LIN {X -0.026,Y -170.982,Z 961.915,A 0.000,B 0.000,C 90.000,E1 344.685} C_DIS
LIN {X 0.007,Y -175.624,Z 961.891,A 0.000,B 0.000,C 90.000,E1 340.369} C_DIS
LIN {X -0.036,Y -180.192,Z 961.872,A 0.000,B 0.000,C 90.000,E1 336.975} C_DIS
LIN {X 0.007,Y -185.517,Z 961.853,A 0.000,B 0.000,C 90.000,E1 333.589} C_DIS
LIN {X 0.016,Y -191.502,Z 961.835,A 0.000,B 0.000,C 90.000,E1 330.255} C_DIS
LIN {X 0.044,Y -198.134,Z 961.817,A 0.000,B 0.000,C 90.000,E1 326.962} C_DIS
LIN {X -0.044,Y -205.288,Z 961.799,A 0.000,B 0.000,C 90.000,E1 323.749} C_DIS
LIN {X 0.027,Y -214.038,Z 961.779,A 0.000,B 0.000,C 90.000,E1 320.150} C_DIS
LIN {X -0.039,Y -223.598,Z 961.759,A 0.000,B 0.000,C 90.000,E1 316.662} C_DIS
LIN {X 0.117,Y -231.821,Z 961.744,A 0.000,B 0.000,C 90.000,E1 313.947} C_DIS
LIN {X 0.013,Y -239.745,Z 961.732,A 0.000,B 0.000,C 90.000,E1 311.714} C_DIS
LIN {X 0.060,Y -248.525,Z 961.719,A 0.000,B 0.000,C 90.000,E1 309.483} C_DIS
LIN {X -0.009,Y -258.437,Z 961.707,A 0.000,B 0.000,C 90.000,E1 307.317} C_DIS
LIN {X 0.026,Y -271.478,Z 961.693,A 0.000,B 0.000,C 90.000,E1 304.818} C_DIS
LIN {X -0.029,Y -289.720,Z 961.676,A 0.000,B 0.000,C 90.000,E1 301.720} C_DIS
LIN {X 0.062,Y -307.259,Z 961.661,A 0.000,B 0.000,C 90.000,E1 299.027} C_DIS
LIN {X 0.052,Y -321.608,Z 961.651,A 0.000,B 0.000,C 90.000,E1 297.078} C_DIS
LIN {X -0.075,Y -337.425,Z 961.640,A 0.000,B 0.000,C 90.000,E1 295.207} C_DIS
LIN {X 0.054,Y -361.602,Z 961.626,A 0.000,B 0.000,C 90.000,E1 292.589} C_DIS
LIN {X 0.114,Y -380.487,Z 961.615,A 0.000,B 0.000,C 90.000,E1 290.684} C_DIS
LIN {X -0.082,Y -396.466,Z 961.606,A 0.000,B 0.000,C 90.000,E1 289.141} C_DIS
LIN {X -0.088,Y -406.784,Z 961.601,A 0.000,B 0.000,C 90.000,E1 288.109} C_DIS
LIN {X -0.044,Y -416.963,Z 961.595,A 0.000,B 0.000,C 90.000,E1 287.040} C_DIS
LIN {X -0.041,Y -426.720,Z 961.589,A 0.000,B 0.000,C 90.000,E1 285.969} C_DIS
LIN {X -0.090,Y -435.970,Z 961.583,A 0.000,B 0.000,C 90.000,E1 284.898} C_DIS
LIN {X -0.032,Y -444.624,Z 961.577,A 0.000,B 0.000,C 90.000,E1 283.828} C_DIS
LIN {X 0.023,Y -452.841,Z 961.571,A 0.000,B 0.000,C 90.000,E1 282.771} C_DIS
LIN {X 0.004,Y -462.674,Z 961.564,A 0.000,B 0.000,C 90.000,E1 281.478} C_DIS
LIN {X 0.188,Y -470.065,Z 961.558,A 0.000,B 0.000,C 90.000,E1 280.433} C_DIS
LIN {X 0.219,Y -475.061,Z 961.554,A 0.000,B 0.000,C 90.000,E1 279.670} C_DIS
LIN {X 0.205,Y -479.402,Z 961.550,A 0.000,B 0.000,C 90.000,E1 278.916} C_DIS
LIN {X 0.234,Y -483.153,Z 961.545,A 0.000,B 0.000,C 90.000,E1 278.163} C_DIS
LIN {X -0.191,Y -486.193,Z 961.541,A 0.000,B 0.000,C 90.000,E1 277.466} C_DIS
LIN {X -0.004,Y -487.783,Z 961.539,A 0.000,B 0.000,C 90.000,E1 276.947} C_DIS
LIN {X 0.195,Y -489.108,Z 961.536,A 0.000,B 0.000,C 90.000,E1 276.429} C_DIS
LIN {X -0.083,Y -490.089,Z 961.533,A 0.000,B 0.000,C 90.000,E1 275.967} C_DIS
LIN {X 0.087,Y -490.692,Z 961.530,A 0.000,B 0.000,C 90.000,E1 275.454} C_DIS
LIN {X -0.177,Y -490.975,Z 961.528,A 0.000,B 0.000,C 90.000,E1 274.992} C_DIS
LIN {X 0.048,Y -490.856,Z 961.525,A 0.000,B 0.000,C 90.000,E1 274.473} C_DIS
LIN {X -0.216,Y -490.241,Z 961.522,A 0.000,B 0.000,C 90.000,E1 274.012} C_DIS
LIN {X -0.024,Y -489.133,Z 961.519,A 0.000,B 0.000,C 90.000,E1 273.498} C_DIS
LIN {X 0.191,Y -487.457,Z 961.517,A 0.000,B 0.000,C 90.000,E1 272.980} C_DIS
LIN {X -0.110,Y -485.167,Z 961.514,A 0.000,B 0.000,C 90.000,E1 272.522} C_DIS
LIN {X 0.061,Y -482.109,Z 961.511,A 0.000,B 0.000,C 90.000,E1 272.007} C_DIS
LIN {X 0.230,Y -478.218,Z 961.508,A 0.000,B 0.000,C 90.000,E1 271.489} C_DIS
LIN {X -0.113,Y -473.302,Z 961.506,A 0.000,B 0.000,C 90.000,E1 271.031} C_DIS
LIN {X 0.122,Y -467.447,Z 961.503,A 0.000,B 0.000,C 90.000,E1 270.516} C_DIS
LIN {X -0.094,Y -461.291,Z 961.501,A 0.000,B 0.000,C 90.000,E1 270.115} C_DIS
LIN {X 0.113,Y -454.819,Z 961.498,A 0.000,B 0.000,C 90.000,E1 269.714} C_DIS
LIN {X -0.166,Y -447.990,Z 961.497,A 0.000,B 0.000,C 90.000,E1 269.427} C_DIS
LIN {X -0.029,Y -441.097,Z 961.495,A 0.000,B 0.000,C 90.000,E1 269.141} C_DIS
LIN {X -0.002,Y -433.778,Z 961.494,A 0.000,B 0.000,C 90.000,E1 268.912} C_DIS
LIN {X -0.186,Y -422.204,Z 961.493,A 0.000,B 0.000,C 90.000,E1 268.682} C_DIS
LIN {X 0.177,Y -413.488,Z 961.492,A 0.000,B 0.000,C 90.000,E1 268.511} C_DIS
LIN {X 0.087,Y -402.266,Z 961.491,A 0.000,B 0.000,C 90.000,E1 268.453} C_DIS
LIN {X 0.012,Y -181.206,Z 961.491,A 0.000,B 0.000,C 90.000,E1 268.453} C_DIS
LIN {X -0.069,Y -180.871,Z 961.472,A 0.000,B 0.000,C 90.000,E1 265.065} C_DIS
LIN {X -0.011,Y -178.987,Z 961.444,A 0.000,B 0.000,C 90.000,E1 259.982} C_DIS
LIN {X 0.000,Y -177.967,Z 961.435,A 0.000,B 0.000,C 90.000,E1 258.285} C_DIS
LIN {X 0.018,Y -175.611,Z 961.411,A 0.000,B 0.000,C 90.000,E1 254.031} C_DIS
LIN {X 0.031,Y -172.332,Z 961.388,A 0.000,B 0.000,C 90.000,E1 249.752} C_DIS
LIN {X 0.009,Y -171.809,Z 961.383,A 0.000,B 0.000,C 90.000,E1 248.901} C_DIS
LIN {X 0.017,Y -170.271,Z 961.373,A 0.000,B 0.000,C 90.000,E1 247.177} C_DIS
LIN {X -0.047,Y -166.813,Z 961.349,A 0.000,B 0.000,C 90.000,E1 242.871} C_DIS
LIN {X 0.011,Y -162.794,Z 961.325,A 0.000,B 0.000,C 90.000,E1 238.486} C_DIS
LIN {X 0.071,Y -161.482,Z 961.315,A 0.000,B 0.000,C 90.000,E1 236.707} C_DIS
LIN {X -0.014,Y -157.478,Z 961.291,A 0.000,B 0.000,C 90.000,E1 232.316} C_DIS
LIN {X 0.044,Y -155.494,Z 961.276,A 0.000,B 0.000,C 90.000,E1 229.622} C_DIS
LIN {X -0.024,Y -151.800,Z 961.251,A 0.000,B 0.000,C 90.000,E1 225.162} C_DIS
LIN {X -0.012,Y -150.009,Z 961.236,A 0.000,B 0.000,C 90.000,E1 222.447} C_DIS
LIN {X 0.020,Y -146.835,Z 961.211,A 0.000,B 0.000,C 90.000,E1 217.890} C_DIS
LIN {X 0.006,Y -145.417,Z 961.195,A 0.000,B 0.000,C 90.000,E1 215.152} C_DIS
LIN {X 0.041,Y -142.845,Z 961.170,A 0.000,B 0.000,C 90.000,E1 210.541} C_DIS
LIN {X -0.028,Y -141.459,Z 961.149,A 0.000,B 0.000,C 90.000,E1 206.873} C_DIS
LIN {X 0.011,Y -139.374,Z 961.113,A 0.000,B 0.000,C 90.000,E1 200.355} C_DIS
LIN {X -0.047,Y -138.825,Z 961.098,A 0.000,B 0.000,C 90.000,E1 197.583} C_DIS
LIN {X 0.042,Y -138.353,Z 961.056,A 0.000,B 0.000,C 90.000,E1 190.074} C_DIS
LIN {X 0.015,Y -139.531,Z 961.004,A 0.000,B 0.000,C 90.000,E1 180.745} C_DIS
LIN {X -0.032,Y -141.210,Z 960.973,A 0.000,B 0.000,C 90.000,E1 175.179} C_DIS
LIN {X 0.068,Y -142.585,Z 960.958,A 0.000,B 0.000,C 90.000,E1 172.356} C_DIS
LIN {X 0.022,Y -144.882,Z 960.932,A 0.000,B 0.000,C 90.000,E1 167.757} C_DIS
LIN {X -0.024,Y -147.509,Z 960.912,A 0.000,B 0.000,C 90.000,E1 164.102} C_DIS
LIN {X 0.050,Y -150.102,Z 960.891,A 0.000,B 0.000,C 90.000,E1 160.423} C_DIS
LIN {X 0.063,Y -153.459,Z 960.871,A 0.000,B 0.000,C 90.000,E1 156.794} C_DIS
LIN {X -0.086,Y -157.822,Z 960.846,A 0.000,B 0.000,C 90.000,E1 152.359} C_DIS
LIN {X -0.054,Y -162.105,Z 960.827,A 0.000,B 0.000,C 90.000,E1 148.791} C_DIS
LIN {X -0.029,Y -166.306,Z 960.807,A 0.000,B 0.000,C 90.000,E1 145.261} C_DIS
LIN {X -0.034,Y -171.323,Z 960.788,A 0.000,B 0.000,C 90.000,E1 141.778} C_DIS
LIN {X 0.001,Y -176.223,Z 960.768,A 0.000,B 0.000,C 90.000,E1 138.324} C_DIS
LIN {X -0.005,Y -180.502,Z 960.754,A 0.000,B 0.000,C 90.000,E1 135.769} C_DIS
LIN {X -0.024,Y -185.905,Z 960.736,A 0.000,B 0.000,C 90.000,E1 132.405} C_DIS
LIN {X 0.036,Y -190.533,Z 960.722,A 0.000,B 0.000,C 90.000,E1 129.886} C_DIS
LIN {X 0.043,Y -194.856,Z 960.708,A 0.000,B 0.000,C 90.000,E1 127.363} C_DIS
LIN {X 0.012,Y -298.138,Z 960.708,A 0.000,B 0.000,C 90.000,E1 127.363} C_DIS
LIN {X 0.055,Y -303.603,Z 960.706,A 0.000,B 0.000,C 90.000,E1 127.156} C_DIS
LIN {X -0.090,Y -306.032,Z 960.705,A 0.000,B 0.000,C 90.000,E1 126.996} C_DIS
LIN {X 0.108,Y -309.310,Z 960.703,A 0.000,B 0.000,C 90.000,E1 126.583} C_DIS
LIN {X -0.032,Y -311.260,Z 960.702,A 0.000,B 0.000,C 90.000,E1 126.297} C_DIS
LIN {X 0.081,Y -312.785,Z 960.700,A 0.000,B 0.000,C 90.000,E1 125.964} C_DIS
LIN {X 0.057,Y -314.038,Z 960.698,A 0.000,B 0.000,C 90.000,E1 125.644} C_DIS
LIN {X -0.043,Y -325.676,Z 960.678,A 0.000,B 0.000,C 90.000,E1 122.133} C_DIS
LIN {X 0.067,Y -336.594,Z 960.663,A 0.000,B 0.000,C 90.000,E1 119.283} C_DIS
LIN {X 0.171,Y -348.902,Z 960.647,A 0.000,B 0.000,C 90.000,E1 116.488} C_DIS
LIN {X -0.163,Y -362.702,Z 960.632,A 0.000,B 0.000,C 90.000,E1 113.823} C_DIS
LIN {X 0.161,Y -376.325,Z 960.619,A 0.000,B 0.000,C 90.000,E1 111.408} C_DIS
LIN {X -0.151,Y -391.324,Z 960.606,A 0.000,B 0.000,C 90.000,E1 109.141} C_DIS
LIN {X 0.017,Y -407.805,Z 960.594,A 0.000,B 0.000,C 90.000,E1 106.858} C_DIS
LIN {X -0.015,Y -425.886,Z 960.581,A 0.000,B 0.000,C 90.000,E1 104.662} C_DIS
LIN {X 0.021,Y -445.508,Z 960.570,A 0.000,B 0.000,C 90.000,E1 102.535} C_DIS
LIN {X -0.178,Y -468.236,Z 960.557,A 0.000,B 0.000,C 90.000,E1 100.366} C_DIS
LIN {X 0.211,Y -470.122,Z 960.556,A 0.000,B 0.000,C 90.000,E1 100.074} C_DIS
LIN {X 0.057,Y -471.551,Z 960.555,A 0.000,B 0.000,C 90.000,E1 99.849} C_DIS
LIN {X 0.233,Y -473.463,Z 960.552,A 0.000,B 0.000,C 90.000,E1 99.321} C_DIS
LIN {X -0.128,Y -474.266,Z 960.549,A 0.000,B 0.000,C 90.000,E1 98.859} C_DIS
LIN {X -0.006,Y -474.096,Z 960.546,A 0.000,B 0.000,C 90.000,E1 98.341} C_DIS
LIN {X 0.186,Y -472.934,Z 960.544,A 0.000,B 0.000,C 90.000,E1 97.814} C_DIS
LIN {X -0.018,Y -471.927,Z 960.542,A 0.000,B 0.000,C 90.000,E1 97.587} C_DIS
LIN {X -0.157,Y -470.573,Z 960.541,A 0.000,B 0.000,C 90.000,E1 97.352} C_DIS
LIN {X -0.099,Y -458.837,Z 960.531,A 0.000,B 0.000,C 90.000,E1 95.568} C_DIS
LIN {X 0.180,Y -447.158,Z 960.521,A 0.000,B 0.000,C 90.000,E1 93.726} C_DIS
LIN {X -0.098,Y -433.765,Z 960.509,A 0.000,B 0.000,C 90.000,E1 91.661} C_DIS
LIN {X 0.069,Y -416.507,Z 960.493,A 0.000,B 0.000,C 90.000,E1 88.682} C_DIS
LIN {X -0.209,Y -407.500,Z 960.484,A 0.000,B 0.000,C 90.000,E1 87.078} C_DIS
LIN {X -0.139,Y -396.770,Z 960.473,A 0.000,B 0.000,C 90.000,E1 85.122} C_DIS
LIN {X 0.091,Y -385.963,Z 960.462,A 0.000,B 0.000,C 90.000,E1 83.109} C_DIS
LIN {X 0.160,Y -376.480,Z 960.452,A 0.000,B 0.000,C 90.000,E1 81.376} C_DIS
LIN {X 0.112,Y -366.676,Z 960.443,A 0.000,B 0.000,C 90.000,E1 79.634} C_DIS
LIN {X -0.042,Y -356.704,Z 960.433,A 0.000,B 0.000,C 90.000,E1 77.881} C_DIS
LIN {X -0.022,Y -343.236,Z 960.419,A 0.000,B 0.000,C 90.000,E1 75.463} C_DIS
LIN {X -0.013,Y -325.933,Z 960.400,A 0.000,B 0.000,C 90.000,E1 72.054} C_DIS
LIN {X -0.042,Y -313.795,Z 960.386,A 0.000,B 0.000,C 90.000,E1 69.518} C_DIS
LIN {X 0.055,Y -303.278,Z 960.374,A 0.000,B 0.000,C 90.000,E1 67.230} C_DIS
LIN {X 0.034,Y -291.383,Z 960.359,A 0.000,B 0.000,C 90.000,E1 64.588} C_DIS
LIN {X 0.012,Y -281.073,Z 960.346,A 0.000,B 0.000,C 90.000,E1 62.231} C_DIS
LIN {X 0.151,Y -270.810,Z 960.332,A 0.000,B 0.000,C 90.000,E1 59.793} C_DIS
LIN {X -0.115,Y -259.503,Z 960.317,A 0.000,B 0.000,C 90.000,E1 57.041} C_DIS
LIN {X -0.006,Y -247.321,Z 960.299,A 0.000,B 0.000,C 90.000,E1 53.783} C_DIS
LIN {X -0.046,Y -236.137,Z 960.280,A 0.000,B 0.000,C 90.000,E1 50.481} C_DIS
LIN {X 0.065,Y -225.747,Z 960.262,A 0.000,B 0.000,C 90.000,E1 47.067} C_DIS
LIN {X -0.042,Y -217.126,Z 960.245,A 0.000,B 0.000,C 90.000,E1 44.028} C_DIS
LIN {X -0.031,Y -208.998,Z 960.227,A 0.000,B 0.000,C 90.000,E1 40.906} C_DIS
LIN {X -0.022,Y -201.490,Z 960.210,A 0.000,B 0.000,C 90.000,E1 37.729} C_DIS
LIN {X 0.043,Y -194.610,Z 960.192,A 0.000,B 0.000,C 90.000,E1 34.485} C_DIS
LIN {X 0.044,Y -188.375,Z 960.173,A 0.000,B 0.000,C 90.000,E1 31.209} C_DIS
LIN {X 0.018,Y -182.888,Z 960.155,A 0.000,B 0.000,C 90.000,E1 27.897} C_DIS
LIN {X 0.082,Y -178.025,Z 960.136,A 0.000,B 0.000,C 90.000,E1 24.515} C_DIS
LIN {X -0.039,Y -172.973,Z 960.113,A 0.000,B 0.000,C 90.000,E1 20.301} C_DIS
LIN {X 0.053,Y -169.051,Z 960.089,A 0.000,B 0.000,C 90.000,E1 15.969} C_DIS
END
